(* IEC 61131-3 sources: SmartHomeNew/ (part 14) *)

(* ---- PRG_Output_Freshness_Governor.st ---- *)
PROGRAM PRG_Output_Freshness_Governor
VAR
    L_Now_MS : UDINT;
    L_Delta_MS : UDINT;
    L_Output_Valid : BOOL := TRUE;
    L_Error_Code : UDINT := 0;
    L_Error_Text : STRING(160) := '';
END_VAR

L_Now_MS := GVL_STATUS.G_System_Time_MS;
L_Output_Valid := TRUE;
L_Error_Code := 0;
L_Error_Text := '';

IF NOT GVL_RUNTIME_EPOCH.Runtime_Runtime_Barrier_OK THEN
    L_Output_Valid := FALSE;
    L_Error_Code := 6000;
    L_Error_Text := 'Output runtime authority invalid';
END_IF;

IF L_Output_Valid AND (NOT GVL_RUNTIME_EPOCH.Runtime_IO_Publication_Allowed) THEN
    L_Output_Valid := FALSE;
    L_Error_Code := 6001;
    L_Error_Text := 'Output publication not allowed';
END_IF;

IF L_Output_Valid AND (NOT GVL_RUNTIME_SNAPSHOT.Snapshot_Frozen) THEN
    L_Output_Valid := FALSE;
    L_Error_Code := 6100;
    L_Error_Text := 'Runtime snapshot not frozen';
END_IF;

IF L_Output_Valid AND (NOT GVL_RUNTIME_SNAPSHOT.Snapshot_Publication_Allowed) THEN
    L_Output_Valid := FALSE;
    L_Error_Code := 6101;
    L_Error_Text := 'Snapshot publication blocked';
END_IF;

IF L_Output_Valid AND (NOT GVL_RUNTIME_SNAPSHOT.Snapshot_Copy_Valid) THEN
    L_Output_Valid := FALSE;
    L_Error_Code := 6102;
    L_Error_Text := 'Snapshot copy invalid';
END_IF;

IF L_Output_Valid AND (NOT GVL_RUNTIME_SNAPSHOT.Snapshot_Isolation_Valid) THEN
    L_Output_Valid := FALSE;
    L_Error_Code := 6103;
    L_Error_Text := 'Snapshot isolation invalid';
END_IF;

IF L_Output_Valid AND GVL_RUNTIME_SNAPSHOT.Snapshot_Mutation_Detected THEN
    L_Output_Valid := FALSE;
    L_Error_Code := 6104;
    L_Error_Text := 'Snapshot mutation detected';
END_IF;

IF L_Output_Valid AND GVL_DISTRIBUTED_EPOCH.Distributed_Quarantine_Active THEN
    L_Output_Valid := FALSE;
    L_Error_Code := 6200;
    L_Error_Text := 'Distributed reconciliation quarantine active';
END_IF;

IF L_Output_Valid AND (NOT GVL_DISTRIBUTED_SNAPSHOT.Distributed_Publication_Reconciled) THEN
    L_Output_Valid := FALSE;
    L_Error_Code := 6300;
    L_Error_Text := 'Distributed publication reconciliation invalid';
END_IF;

IF L_Output_Valid AND (NOT GVL_DISTRIBUTED_SNAPSHOT.Distributed_Publication_Freeze_Valid) THEN
    L_Output_Valid := FALSE;
    L_Error_Code := 6301;
    L_Error_Text := 'Distributed publication freeze invalid';
END_IF;

IF L_Output_Valid AND (NOT GVL_DISTRIBUTED_SNAPSHOT.Distributed_Snapshot_Consistent) THEN
    L_Output_Valid := FALSE;
    L_Error_Code := 6302;
    L_Error_Text := 'Distributed immutable snapshot inconsistent';
END_IF;

IF L_Output_Valid AND GVL_DISTRIBUTED_SNAPSHOT.Distributed_Snapshot_Quarantine_Active THEN
    L_Output_Valid := FALSE;
    L_Error_Code := 6306;
    L_Error_Text := 'Distributed immutable snapshot quarantine active';
END_IF;

// Finalized distributed publication continuity.
IF L_Output_Valid AND (NOT GVL_DISTRIBUTED_COMMIT.Distributed_Commit_Valid) THEN
    L_Output_Valid := FALSE;
    L_Error_Code := 6400;
    L_Error_Text := 'Distributed commit invalid';
END_IF;

IF L_Output_Valid AND (NOT GVL_DISTRIBUTED_COMMIT.Publication_Prepare_Valid) THEN
    L_Output_Valid := FALSE;
    L_Error_Code := 6402;
    L_Error_Text := 'Distributed publication prepare invalid';
END_IF;

IF L_Output_Valid AND GVL_DISTRIBUTED_COMMIT.Publication_Commit_Requested
   AND (NOT GVL_DISTRIBUTED_COMMIT.Publication_Commit_Confirmed) THEN
    L_Output_Valid := FALSE;
    L_Error_Code := 6403;
    L_Error_Text := 'Distributed publication commit pending';
END_IF;

IF L_Output_Valid AND GVL_DISTRIBUTED_COMMIT.Peer_Commit_Mismatch THEN
    L_Output_Valid := FALSE;
    L_Error_Code := 6404;
    L_Error_Text := 'Distributed peer commit mismatch';
END_IF;

IF L_Output_Valid AND GVL_DISTRIBUTED_COMMIT.Distributed_Commit_Quarantine_Active THEN
    L_Output_Valid := FALSE;
    L_Error_Code := 6401;
    L_Error_Text := 'Distributed commit quarantine active';
END_IF;

IF L_Output_Valid AND GVL_DISTRIBUTED_COMMIT.Commit_Lease_Expired THEN
    L_Output_Valid := FALSE;
    L_Error_Code := 6405;
    L_Error_Text := 'Distributed commit lease expired';
END_IF;

GVL_OUTPUT_EPOCH.Output_Semantic_Continuity_Warning :=
    (NOT GVL_SEMANTIC_PROGRESS.Semantic_Forward_Progress_Valid)
    OR (NOT GVL_SEMANTIC_PROGRESS.Semantic_Execution_Continuity_OK)
    OR GVL_SEMANTIC_PROGRESS.Semantic_Stagnation_Detected
    OR GVL_SEMANTIC_PROGRESS.Semantic_Replay_Suspected
    OR GVL_SEMANTIC_PROGRESS.Semantic_Livelock_Suspected
    OR GVL_SEMANTIC_PROGRESS.Semantic_Deadlock_Suspected
    OR GVL_SEMANTIC_PROGRESS.Semantic_Progress_Lease_Expired
    OR GVL_SEMANTIC_PROGRESS.Semantic_Progress_Quarantine_Active;

IF L_Output_Valid THEN
    IF GVL_OUTPUT_EPOCH.Output_Runtime_Epoch > GVL_RUNTIME_EPOCH.Runtime_Epoch THEN
        L_Output_Valid := FALSE;
        L_Error_Code := 6002;
        L_Error_Text := 'Output epoch ahead of runtime epoch';
    END_IF;
END_IF;

L_Delta_MS := L_Now_MS - GVL_OUTPUT_EPOCH.Output_Last_Refresh_MS;

IF L_Output_Valid AND GVL_OUTPUT_EPOCH.Output_Lease_Active THEN
    IF L_Delta_MS > GVL_OUTPUT_EPOCH.Output_Lease_Timeout_MS THEN
        L_Output_Valid := FALSE;
        L_Error_Code := 6003;
        L_Error_Text := 'Output lease expired';
    END_IF;
END_IF;

IF L_Output_Valid THEN
    GVL_OUTPUT_EPOCH.Output_Publication_Epoch := GVL_OUTPUT_EPOCH.Output_Publication_Epoch + 1;

    GVL_OUTPUT_EPOCH.Output_Publication_Valid := TRUE;
    GVL_OUTPUT_EPOCH.Output_Lease_Active := TRUE;
    GVL_OUTPUT_EPOCH.Output_Lease_Expired := FALSE;

    GVL_OUTPUT_EPOCH.Output_Runtime_Epoch := GVL_RUNTIME_EPOCH.Runtime_Epoch;
    GVL_OUTPUT_EPOCH.Output_Runtime_Epoch_Valid := TRUE;

    GVL_OUTPUT_EPOCH.Output_Last_Publication_MS := L_Now_MS;
    GVL_OUTPUT_EPOCH.Output_Last_Refresh_MS := L_Now_MS;

    IF GVL_CONVERGENCE.Convergence_Release_Allowed THEN
        GVL_OUTPUT_EPOCH.Output_Stale_Detected := FALSE;
        GVL_OUTPUT_EPOCH.Output_Forced_Safe_Decay := FALSE;
    END_IF;

    GVL_OUTPUT_EPOCH.Output_Last_Error_Code := 0;
    GVL_OUTPUT_EPOCH.Output_Last_Error_Text := '';
ELSE
    GVL_OUTPUT_EPOCH.Output_Publication_Valid := FALSE;
    GVL_OUTPUT_EPOCH.Output_Lease_Expired := TRUE;
    GVL_OUTPUT_EPOCH.Output_Stale_Detected := TRUE;
    GVL_OUTPUT_EPOCH.Output_Forced_Safe_Decay := TRUE;

    GVL_OUTPUT_EPOCH.Output_Last_Invalidation_MS := L_Now_MS;
    GVL_OUTPUT_EPOCH.Output_Last_Error_Code := L_Error_Code;
    GVL_OUTPUT_EPOCH.Output_Last_Error_Text := L_Error_Text;
END_IF;
END_PROGRAM

(* ---- PRG_Peer_Session_Publication.st ---- *)
PROGRAM PRG_Peer_Session_Publication
// ======================================================
// PEER SESSION PUBLICATION
// ======================================================
// Canonical local PLC session export.
//
// Purpose:
// publish normalized runtime/session authority state into
// explicit peer-session transport contract surface.
//
// This layer does NOT:
// - perform network replication
// - perform distributed reconciliation
// - consume remote peer state
//
// Future transport/replication layers may replicate these
// fields to partner PLCs or external HA channels.
// ======================================================

GVL_PEER_SESSION.Remote_Session_Valid :=
    GVL_RUNTIME_EPOCH.Runtime_IO_Publication_Allowed;

GVL_PEER_SESSION.Remote_Last_Refresh_MS :=
    GVL_STATUS.G_System_Time_MS;

GVL_PEER_SESSION.Remote_Runtime_Epoch :=
    GVL_RUNTIME_EPOCH.Runtime_Epoch;

GVL_PEER_SESSION.Remote_Snapshot_Epoch :=
    GVL_RUNTIME_SNAPSHOT.Snapshot_Epoch;

GVL_PEER_SESSION.Remote_Boot_Generation :=
    GVL_TIME_MONOTONIC.Boot_Generation_ID;

GVL_PEER_SESSION.Remote_Fencing_Token :=
    GVL_PLC_FENCING.PLC_Fencing_Token;

GVL_PEER_SESSION.Remote_Publication_Allowed :=
    GVL_OUTPUT_EPOCH.Output_Publication_Allowed;

GVL_PEER_SESSION.Remote_Runtime_Healthy :=
    GVL_RUNTIME_EPOCH.Runtime_Healthy;

// >>> BULK_SYNC_ANCHOR: PRG_Peer_Session_Publication <<<
END_PROGRAM

(* ---- PRG_Physical_Deadlock_Resolution_Governor.st ---- *)
PROGRAM PRG_Physical_Deadlock_Resolution_Governor
IF GVL_ENERGY_RESURRECTION_BOUNDARY_FABRIC.Energy_Resurrection_Boundary_Granted
AND NOT GVL_PHYSICAL_DEADLOCK_RESOLUTION_FABRIC.Physical_CircularWait_Detected
AND NOT GVL_PHYSICAL_DEADLOCK_RESOLUTION_FABRIC.CrossDomain_Progress_Deadlock
AND NOT GVL_PHYSICAL_DEADLOCK_RESOLUTION_FABRIC.Recovery_Livelock_Detected
AND NOT GVL_PHYSICAL_DEADLOCK_RESOLUTION_FABRIC.Physical_Progress_Stall_Detected THEN

    GVL_PHYSICAL_DEADLOCK_RESOLUTION_FABRIC.Physical_Deadlock_Resolution_Valid := TRUE;
    GVL_PHYSICAL_DEADLOCK_RESOLUTION_FABRIC.Physical_Deadlock_Resolution_Granted := TRUE;
    GVL_PHYSICAL_DEADLOCK_RESOLUTION_FABRIC.Deadlock_Resolution_Canonical := TRUE;
    GVL_PHYSICAL_DEADLOCK_RESOLUTION_FABRIC.Physical_Forward_Progress_Valid := TRUE;
    GVL_PHYSICAL_DEADLOCK_RESOLUTION_FABRIC.CrossDomain_Execution_Progress_Stable := TRUE;
END_IF;
END_PROGRAM

(* ---- PRG_Physical_Reality_Validation_Governor.st ---- *)
PROGRAM PRG_Physical_Reality_Validation_Governor
// PASSIVE PHYSICS REALITY VERIFICATION
// NO EXECUTION MUTATION
// NO ACTUATION MUTATION
// NO AUTHORITY MUTATION

GVL_PHYSICAL_REALITY_VERIFICATION_FABRIC.Physical_Runtime_Reality_Valid :=
    GVL_OPERATIONAL_INTELLIGENCE_FABRIC.Runtime_Causal_Projection_Valid;

GVL_PHYSICAL_REALITY_VERIFICATION_FABRIC.Commanded_State_Verified_Physically :=
    GVL_RUNTIME_TRANSITION_SYSTEM.Runtime_Transition_Legal;

GVL_PHYSICAL_REALITY_VERIFICATION_FABRIC.Physical_Response_Coherent :=
    GVL_TEMPORAL_CAUSALITY_CLOSURE_FABRIC.Temporal_Causality_Coherent;

GVL_PHYSICAL_REALITY_VERIFICATION_FABRIC.Sensor_Physics_Coherent := TRUE;

IF GVL_RUNTIME_TRANSITION_SYSTEM.Illegal_Runtime_Transition_Observed THEN
    GVL_PHYSICAL_REALITY_VERIFICATION_FABRIC.Physical_Reality_Divergence_Detected := TRUE;
END_IF;

IF GVL_RUNTIME_TRANSITION_SYSTEM.Unsafe_State_Promotion_Observed THEN
    GVL_PHYSICAL_REALITY_VERIFICATION_FABRIC.Commanded_State_Mismatch_Detected := TRUE;
END_IF;

IF GVL_TEMPORAL_CAUSALITY_CLOSURE_FABRIC.Temporal_Fork_Detected THEN
    GVL_PHYSICAL_REALITY_VERIFICATION_FABRIC.Impossible_Physical_Response_Detected := TRUE;
END_IF;

END_PROGRAM

(* ---- PRG_Physical_SafeState_Lattice_Governor.st ---- *)
PROGRAM PRG_Physical_SafeState_Lattice_Governor
VAR
    L_Now_MS : UDINT;
    L_Valid : BOOL := TRUE;
END_VAR

L_Now_MS := GVL_STATUS.G_System_Time_MS;

GVL_PHYSICAL_SAFESTATE_LATTICE_FABRIC.Physical_SafeState_Lattice_Valid := FALSE;
GVL_PHYSICAL_SAFESTATE_LATTICE_FABRIC.Physical_SafeState_Lattice_Granted := FALSE;
GVL_PHYSICAL_SAFESTATE_LATTICE_FABRIC.Physical_SafeState_Lattice_Quarantine_Active := TRUE;

IF NOT GVL_GOVERNANCE_PUBLICATION_BINDING_FABRIC.Governance_Publication_Binding_Granted THEN
    L_Valid := FALSE;
END_IF;

IF GVL_PHYSICAL_SAFESTATE_LATTICE_FABRIC.SafeState_Ambiguity_Detected
OR GVL_PHYSICAL_SAFESTATE_LATTICE_FABRIC.Partial_SafeState_Asymmetry_Detected
OR GVL_PHYSICAL_SAFESTATE_LATTICE_FABRIC.Physical_SafeState_Deadlock_Detected
OR GVL_PHYSICAL_SAFESTATE_LATTICE_FABRIC.Unsafe_SafeState_Topology_Detected
OR GVL_PHYSICAL_SAFESTATE_LATTICE_FABRIC.Residual_Unsafe_Actuation_Detected
OR GVL_PHYSICAL_SAFESTATE_LATTICE_FABRIC.SafeState_Energy_Leakage_Detected THEN
    L_Valid := FALSE;
END_IF;

IF L_Valid THEN
    GVL_PHYSICAL_SAFESTATE_LATTICE_FABRIC.Physical_SafeState_Lattice_Valid := TRUE;
    GVL_PHYSICAL_SAFESTATE_LATTICE_FABRIC.Physical_SafeState_Lattice_Granted := TRUE;
    GVL_PHYSICAL_SAFESTATE_LATTICE_FABRIC.Physical_SafeState_Lattice_Quarantine_Active := FALSE;

    GVL_PHYSICAL_SAFESTATE_LATTICE_FABRIC.Canonical_SafeState_Topology_Valid := TRUE;
    GVL_PHYSICAL_SAFESTATE_LATTICE_FABRIC.Physical_SafeState_Lattice_Coherent := TRUE;
    GVL_PHYSICAL_SAFESTATE_LATTICE_FABRIC.Deterministic_FailSafe_Convergence_Granted := TRUE;

    GVL_PHYSICAL_SAFESTATE_LATTICE_FABRIC.Physical_SafeState_Lattice_Epoch :=
        GVL_GOVERNANCE_PUBLICATION_BINDING_FABRIC.Governance_Publication_Binding_Epoch;

    GVL_PHYSICAL_SAFESTATE_LATTICE_FABRIC.Physical_SafeState_Lattice_Epoch_Coherent := TRUE;
    GVL_PHYSICAL_SAFESTATE_LATTICE_FABRIC.Physical_SafeState_Lattice_Last_Update_MS := L_Now_MS;
    GVL_PHYSICAL_SAFESTATE_LATTICE_FABRIC.Physical_SafeState_Lattice_Lease_Expired := FALSE;
END_IF;

END_PROGRAM

(* ---- PRG_Physical_Snapshot_Governor.st ---- *)
PROGRAM PRG_Physical_Snapshot_Governor
VAR
    L_Now_MS : UDINT;
    L_Snapshot_Valid : BOOL := TRUE;
    L_Error_Code : UDINT := 0;
    L_Error_Text : STRING(160) := '';
END_VAR

L_Now_MS := GVL_STATUS.G_System_Time_MS;
L_Snapshot_Valid := TRUE;
L_Error_Code := 0;
L_Error_Text := '';

GVL_PHYSICAL_SNAPSHOT.Physical_Snapshot_Valid := FALSE;
GVL_PHYSICAL_SNAPSHOT.Physical_Snapshot_Frozen := FALSE;
GVL_PHYSICAL_SNAPSHOT.Physical_Snapshot_Publication_Allowed := FALSE;
GVL_PHYSICAL_SNAPSHOT.Physical_Snapshot_Isolation_Valid := FALSE;
GVL_PHYSICAL_SNAPSHOT.Physical_Snapshot_Copy_Valid := FALSE;
GVL_PHYSICAL_SNAPSHOT.Physical_Snapshot_Freshness_Valid := FALSE;
GVL_PHYSICAL_SNAPSHOT.Physical_Snapshot_Consensus_Coherent := FALSE;
GVL_PHYSICAL_SNAPSHOT.Physical_Snapshot_Causality_Coherent := FALSE;

GVL_PHYSICAL_SNAPSHOT.Physical_Snapshot_Runtime_Epoch := ULINT_TO_UDINT(GVL_RUNTIME_EPOCH.Runtime_Epoch);
GVL_PHYSICAL_SNAPSHOT.Physical_Snapshot_Output_Epoch := ULINT_TO_UDINT(GVL_OUTPUT_EPOCH.Output_Publication_Epoch);

IF NOT GVL_RUNTIME_EPOCH.Runtime_Runtime_Barrier_OK THEN
    L_Snapshot_Valid := FALSE;
    L_Error_Code := 23000;
    L_Error_Text := 'Physical snapshot runtime barrier invalid';
END_IF;

IF L_Snapshot_Valid AND NOT GVL_OUTPUT_EPOCH.Output_Publication_Valid THEN
    L_Snapshot_Valid := FALSE;
    L_Error_Code := 23001;
    L_Error_Text := 'Physical snapshot output publication invalid';
END_IF;

IF L_Snapshot_Valid AND GVL_PHYSICAL_SNAPSHOT.Physical_Snapshot_Mutation_Detected THEN
    L_Snapshot_Valid := FALSE;
    L_Error_Code := 23002;
    L_Error_Text := 'Physical snapshot mutation detected';
END_IF;

IF L_Snapshot_Valid AND GVL_PHYSICAL_SNAPSHOT.Physical_Snapshot_Replay_Suspected THEN
    L_Snapshot_Valid := FALSE;
    L_Error_Code := 23003;
    L_Error_Text := 'Physical snapshot replay suspected';
END_IF;

IF L_Snapshot_Valid AND GVL_PHYSICAL_SNAPSHOT.Physical_Snapshot_Lease_Expired THEN
    L_Snapshot_Valid := FALSE;
    L_Error_Code := 23004;
    L_Error_Text := 'Physical snapshot lease expired';
END_IF;

IF L_Snapshot_Valid THEN
    GVL_PHYSICAL_SNAPSHOT.Physical_Snapshot_Valid := TRUE;
    GVL_PHYSICAL_SNAPSHOT.Physical_Snapshot_Frozen := TRUE;
    GVL_PHYSICAL_SNAPSHOT.Physical_Snapshot_Publication_Allowed := TRUE;
    GVL_PHYSICAL_SNAPSHOT.Physical_Snapshot_Isolation_Valid := TRUE;
    GVL_PHYSICAL_SNAPSHOT.Physical_Snapshot_Copy_Valid := TRUE;
    GVL_PHYSICAL_SNAPSHOT.Physical_Snapshot_Freshness_Valid := TRUE;
    GVL_PHYSICAL_SNAPSHOT.Physical_Snapshot_Consensus_Coherent := TRUE;
    GVL_PHYSICAL_SNAPSHOT.Physical_Snapshot_Causality_Coherent := TRUE;
    GVL_PHYSICAL_SNAPSHOT.Physical_Snapshot_Epoch := GVL_PHYSICAL_SNAPSHOT.Physical_Snapshot_Epoch + 1;
    GVL_PHYSICAL_SNAPSHOT.Physical_Snapshot_Last_Update_MS := L_Now_MS;
    GVL_PHYSICAL_SNAPSHOT.Physical_Snapshot_Last_Error_Code := 0;
    GVL_PHYSICAL_SNAPSHOT.Physical_Snapshot_Last_Error_Text := '';
ELSE
    GVL_PHYSICAL_SNAPSHOT.Physical_Snapshot_Valid := FALSE;
    GVL_PHYSICAL_SNAPSHOT.Physical_Snapshot_Frozen := FALSE;
    GVL_PHYSICAL_SNAPSHOT.Physical_Snapshot_Publication_Allowed := FALSE;
    GVL_PHYSICAL_SNAPSHOT.Physical_Snapshot_Last_Error_Code := L_Error_Code;
    GVL_PHYSICAL_SNAPSHOT.Physical_Snapshot_Last_Error_Text := L_Error_Text;
    GVL_PHYSICAL_SNAPSHOT.Physical_Snapshot_Invalidation_Count := GVL_PHYSICAL_SNAPSHOT.Physical_Snapshot_Invalidation_Count + 1;
END_IF;

END_PROGRAM

(* ---- PRG_PLC_Arbitration.st ---- *)
PROGRAM PRG_PLC_Arbitration
// Local-only PLC authority for the cold-spare architecture.
//
// Hot A/B failover and lowest-ID arbitration are intentionally disabled.
// The reserve PLC is not expected to be connected to the same physical outputs
// during normal runtime.

GVL_STATUS.G_Is_Active_PLC := TRUE;
GVL_STATUS.G_Other_PLC_Is_Active := FALSE;
GVL_STATUS.G_Remote_PLC_Alive := FALSE;
GVL_STATUS.G_Active_PLC_ID := GVL_STATUS.G_Local_PLC_ID;

// Keep remote visibility fields reset so old partner pulses cannot resurrect a
// standby/active split-brain path.
GVL_STATUS.G_Remote_PLC_Pulse := FALSE;
GVL_STATUS.G_Remote_PLC_Last_Seen_MS := 0;

// >>> BULK_SYNC_ANCHOR: PRG_PLC_Arbitration <<<
END_PROGRAM

(* ---- PRG_PLC_Fencing_Governor.st ---- *)
PROGRAM PRG_PLC_Fencing_Governor
VAR
    L_Now_MS : UDINT;
END_VAR

L_Now_MS := GVL_STATUS.G_System_Time_MS;

// ======================================================
// LOCAL-ONLY PLC FENCING GOVERNOR
// ======================================================
// Cold-spare architecture: there is exactly one runtime owner.
// A reserve PLC is not connected in parallel and is not allowed to arbitrate
// outputs during normal runtime. Therefore split-brain/stale-owner detection is
// held inactive here while still publishing a valid local ownership epoch/token
// for downstream authority checks.
// ======================================================

GVL_PLC_FENCING.PLC_Heartbeat_Only_Mode := FALSE;
GVL_PLC_FENCING.PLC_Split_Brain_Detected := FALSE;
GVL_PLC_FENCING.PLC_Stale_Owner_Detected := FALSE;
GVL_PLC_FENCING.PLC_Asymmetric_Partition_Detected := FALSE;
GVL_PLC_FENCING.PLC_Forced_Safe_Quarantine := FALSE;

GVL_PLC_FENCING.PLC_Ownership_Epoch := GVL_PLC_FENCING.PLC_Ownership_Epoch + 1;
GVL_PLC_FENCING.PLC_Fencing_Token := GVL_PLC_FENCING.PLC_Ownership_Epoch;

GVL_PLC_FENCING.PLC_Ownership_Valid := TRUE;
GVL_PLC_FENCING.PLC_Semantic_Authority_Valid := TRUE;

GVL_PLC_FENCING.PLC_Lease_Active := TRUE;
GVL_PLC_FENCING.PLC_Lease_Expired := FALSE;
GVL_PLC_FENCING.PLC_Last_Lease_Refresh_MS := L_Now_MS;
GVL_PLC_FENCING.PLC_Last_Authority_Validation_MS := L_Now_MS;

GVL_PLC_FENCING.PLC_Last_Error_Code := 0;
GVL_PLC_FENCING.PLC_Last_Error_Text := '';

// >>> BULK_SYNC_ANCHOR: PRG_PLC_Fencing_Governor <<<
END_PROGRAM

(* ---- PRG_Policy.st ---- *)
PROGRAM PRG_Policy
VAR
    L_Away_Elapsed_MS : UDINT;
    L_Restore_Elapsed_MS : UDINT;
    L_Return_Delta_MS : UDINT;
    L_Return_Grace_Elapsed_MS : UDINT;
    L_Away_Return_Window_Reached : BOOL;
    L_Previous_Away_Active : BOOL := FALSE;
    L_Previous_Away_Level : BYTE := 0;
END_VAR

GVL_POLICY.G_Away_Restore_Requested := FALSE;

// ============================================================
// CONFIGURATION SAFETY CLAMP
// ============================================================
// Configuration validation is diagnostic-only here.
// System mode ownership remains in FB_State_Manager via
// FB_System_Health_Orchestrator. Policy must not directly write
// GVL_STATE.G_System_Mode.
IF GVL_CONFIG_VALIDATION.G_Config_Force_Safe_Mode AND
   (NOT GVL_CONFIG_VALIDATION.G_Config_Valid) AND
   (GVL_STATE.G_System_Mode = E_System_Operating_Mode.MODE_NORMAL) THEN
    GVL_STATUS.G_Diagnostics.Subsystem_Degraded := TRUE;
    GVL_STATUS.G_System_Mode_Text := 'CONFIG DEGRADED';
END_IF;

// ============================================================
// SCENARIO POLICY OWNER
// ============================================================

// 1. Base priority resolution
IF GVL_STATE.G_System_Mode = E_System_Operating_Mode.MODE_SAFE_STOP THEN
    GVL_POLICY.G_Scenario_Intent := E_SCENARIO_TYPE.SCENARIO_NONE;
    GVL_POLICY.G_Scenario_Source := SRC_SAFETY;

ELSIF GVL_POLICY.G_Scenario_Request_Operator <> E_SCENARIO_TYPE.SCENARIO_NONE THEN
    GVL_POLICY.G_Scenario_Intent := GVL_POLICY.G_Scenario_Request_Operator;
    GVL_POLICY.G_Scenario_Source := SRC_OPERATOR;

ELSIF GVL_POLICY.G_Scenario_Request_Gateway <> E_SCENARIO_TYPE.SCENARIO_NONE THEN
    GVL_POLICY.G_Scenario_Intent := GVL_POLICY.G_Scenario_Request_Gateway;
    GVL_POLICY.G_Scenario_Source := SRC_GATEWAY;

ELSIF GVL_POLICY.G_Scenario_Request_Rule <> E_SCENARIO_TYPE.SCENARIO_NONE THEN
    GVL_POLICY.G_Scenario_Intent := GVL_POLICY.G_Scenario_Request_Rule;
    GVL_POLICY.G_Scenario_Source := SRC_RULE;

ELSE
    GVL_POLICY.G_Scenario_Intent := GVL_STATUS.G_Current_Scenario;
    GVL_POLICY.G_Scenario_Source := SRC_NONE;
END_IF;

// 2. Fail-safe clamp
CASE GVL_STATE.G_System_Mode OF
    E_System_Operating_Mode.MODE_SAFE_STOP:
        GVL_POLICY.G_Scenario_Intent := E_SCENARIO_TYPE.SCENARIO_NONE;
        GVL_POLICY.G_Scenario_Source := SRC_SAFETY;

    E_System_Operating_Mode.MODE_FREEZE_PROTECTION:
        GVL_POLICY.G_Scenario_Intent := E_SCENARIO_TYPE.SCENARIO_NONE;
        GVL_POLICY.G_Scenario_Source := SRC_POLICY;

    E_System_Operating_Mode.MODE_DEGRADED:
        CASE GVL_POLICY.G_Scenario_Intent OF
            E_SCENARIO_TYPE.SCENARIO_NONE,
            E_SCENARIO_TYPE.SCENARIO_PRESENCE,
            E_SCENARIO_TYPE.SCENARIO_AWAY,
            E_SCENARIO_TYPE.SCENARIO_SLEEP:
                ;
        ELSE
            GVL_POLICY.G_Scenario_Intent := E_SCENARIO_TYPE.SCENARIO_NONE;
            GVL_POLICY.G_Scenario_Source := SRC_POLICY;
        END_CASE;
END_CASE;

// 3. Context automation
IF GVL_STATE.G_System_Mode = E_System_Operating_Mode.MODE_NORMAL THEN
    IF GVL_ALARM.G_Security_Armed AND
       (GVL_POLICY.G_Scenario_Request_Operator = E_SCENARIO_TYPE.SCENARIO_NONE) AND
       (GVL_POLICY.G_Scenario_Request_Gateway = E_SCENARIO_TYPE.SCENARIO_NONE) AND
       (GVL_POLICY.G_Scenario_Request_Rule = E_SCENARIO_TYPE.SCENARIO_NONE) AND
       (GVL_POLICY.G_Scenario_Intent <> E_SCENARIO_TYPE.SCENARIO_AWAY) THEN
        GVL_POLICY.G_Scenario_Intent := E_SCENARIO_TYPE.SCENARIO_AWAY;
        GVL_POLICY.G_Scenario_Source := SRC_POLICY;
    END_IF;
END_IF;

// 4. Degraded adaptation
IF GVL_STATE.G_System_Mode = E_System_Operating_Mode.MODE_DEGRADED THEN
    IF (GVL_POLICY.G_Scenario_Request_Operator = E_SCENARIO_TYPE.SCENARIO_NONE) AND
       (GVL_POLICY.G_Scenario_Request_Gateway = E_SCENARIO_TYPE.SCENARIO_NONE) AND
       (GVL_POLICY.G_Scenario_Request_Rule = E_SCENARIO_TYPE.SCENARIO_NONE) THEN

        IF GVL_ALARM.G_Security_Armed THEN
            GVL_POLICY.G_Scenario_Intent := E_SCENARIO_TYPE.SCENARIO_AWAY;
            GVL_POLICY.G_Scenario_Source := SRC_POLICY;

        ELSIF GVL_POLICY.G_Scenario_Intent = E_SCENARIO_TYPE.SCENARIO_PRESENCE THEN
            GVL_POLICY.G_Scenario_Intent := E_SCENARIO_TYPE.SCENARIO_SLEEP;
            GVL_POLICY.G_Scenario_Source := SRC_POLICY;
        END_IF;
    END_IF;
END_IF;

// ============================================================
// AWAY LEVEL POLICY
// ============================================================
// 0=none, 1=short, 2=medium, 3=long.
// Short: light 100%, heating -1C, simulation off.
// Medium: light/simulation medium, heating -3C, simulation 0.3.
// Long: minimal reasonable heating economy; planned-return preheat may
// temporarily raise selected rooms before the expected arrival.
L_Away_Return_Window_Reached := FALSE;

IF GVL_POLICY.G_Scenario_Intent = E_SCENARIO_TYPE.SCENARIO_AWAY THEN
    IF NOT GVL_POLICY.G_Away_Active THEN
        GVL_POLICY.G_Away_Active := TRUE;
        GVL_POLICY.G_Away_Start_MS := GVL_TIME_SERVICE.G_Now_MS;
        GVL_POLICY.G_Away_Elapsed_MS := 0;
        GVL_POLICY.G_Away_Level := 1;
        GVL_POLICY.G_Away_Return_Preheat_Active := FALSE;
        GVL_POLICY.G_Away_Return_Grace_Active := FALSE;
        GVL_POLICY.G_Away_Return_Expired := FALSE;
    ELSE
        IF GVL_TIME_SERVICE.G_Now_MS >= GVL_POLICY.G_Away_Start_MS THEN
            L_Away_Elapsed_MS := GVL_TIME_SERVICE.G_Now_MS - GVL_POLICY.G_Away_Start_MS;
        ELSE
            L_Away_Elapsed_MS := (4294967295 - GVL_POLICY.G_Away_Start_MS) + GVL_TIME_SERVICE.G_Now_MS + 1;
        END_IF;

        GVL_POLICY.G_Away_Elapsed_MS := L_Away_Elapsed_MS;

        IF L_Away_Elapsed_MS >= GVL_POLICY.G_Away_Medium_To_Long_MS THEN
            GVL_POLICY.G_Away_Level := 3;
        ELSIF L_Away_Elapsed_MS >= GVL_POLICY.G_Away_Short_To_Medium_MS THEN
            GVL_POLICY.G_Away_Level := 2;
        ELSE
            GVL_POLICY.G_Away_Level := 1;
        END_IF;
    END_IF;

    // Planned return preheat window.
    IF GVL_POLICY.G_Away_Planned_Return_Enabled AND NOT GVL_POLICY.G_Away_Return_Expired THEN
        IF GVL_POLICY.G_Away_Planned_Return_MS >= GVL_TIME_SERVICE.G_Now_MS THEN
            L_Return_Delta_MS := GVL_POLICY.G_Away_Planned_Return_MS - GVL_TIME_SERVICE.G_Now_MS;
            L_Away_Return_Window_Reached := (L_Return_Delta_MS <= GVL_POLICY.G_Away_Preheat_Lead_MS);
        ELSE
            L_Away_Return_Window_Reached := TRUE;
        END_IF;

        IF L_Away_Return_Window_Reached THEN
            GVL_POLICY.G_Away_Return_Preheat_Active := TRUE;

            IF NOT GVL_POLICY.G_Away_Return_Grace_Active THEN
                GVL_POLICY.G_Away_Return_Grace_Active := TRUE;
                GVL_POLICY.G_Away_Return_Grace_Start_MS := GVL_TIME_SERVICE.G_Now_MS;
            END_IF;
        END_IF;

        IF GVL_POLICY.G_Away_Return_Grace_Active THEN
            IF GVL_TIME_SERVICE.G_Now_MS >= GVL_POLICY.G_Away_Return_Grace_Start_MS THEN
                L_Return_Grace_Elapsed_MS := GVL_TIME_SERVICE.G_Now_MS - GVL_POLICY.G_Away_Return_Grace_Start_MS;
            ELSE
                L_Return_Grace_Elapsed_MS := (4294967295 - GVL_POLICY.G_Away_Return_Grace_Start_MS) + GVL_TIME_SERVICE.G_Now_MS + 1;
            END_IF;

            IF L_Return_Grace_Elapsed_MS >= GVL_POLICY.G_Away_Return_Grace_MS THEN
                GVL_POLICY.G_Away_Return_Expired := TRUE;
                GVL_POLICY.G_Away_Return_Preheat_Active := FALSE;
                GVL_POLICY.G_Away_Return_Grace_Active := FALSE;
            END_IF;
        END_IF;
    ELSE
        GVL_POLICY.G_Away_Return_Preheat_Active := FALSE;
        GVL_POLICY.G_Away_Return_Grace_Active := FALSE;
    END_IF;

    CASE GVL_POLICY.G_Away_Level OF
        1:
            GVL_POLICY.G_Away_Simulation_Active := FALSE;
            GVL_POLICY.G_Away_Simulation_Intensity := 0.0;
            GVL_POLICY.G_Away_Heating_Offset_C := -1.0;
        2:
            GVL_POLICY.G_Away_Simulation_Active := TRUE;
            GVL_POLICY.G_Away_Simulation_Intensity := 0.3;
            GVL_POLICY.G_Away_Heating_Offset_C := -3.0;
        3:
            GVL_POLICY.G_Away_Simulation_Active := TRUE;
            GVL_POLICY.G_Away_Simulation_Intensity := 0.2;

            IF GVL_POLICY.G_Away_Return_Preheat_Active THEN
                GVL_POLICY.G_Away_Heating_Offset_C := 0.0;
            ELSE
                GVL_POLICY.G_Away_Heating_Offset_C := GVL_POLICY.G_Away_Long_Economy_Setpoint_C - 22.0;
            END_IF;
    ELSE
            GVL_POLICY.G_Away_Simulation_Active := FALSE;
            GVL_POLICY.G_Away_Simulation_Intensity := 0.0;
            GVL_POLICY.G_Away_Heating_Offset_C := 0.0;
    END_CASE;

ELSE
    IF GVL_POLICY.G_Away_Active AND (GVL_POLICY.G_Away_Level = 1) THEN
        GVL_POLICY.G_Away_Restore_Requested := TRUE;
        GVL_POLICY.G_Away_Restore_Active := TRUE;
        GVL_POLICY.G_Away_Restore_Start_MS := GVL_TIME_SERVICE.G_Now_MS;
    END_IF;

    GVL_POLICY.G_Away_Active := FALSE;
    GVL_POLICY.G_Away_Level := 0;
    GVL_POLICY.G_Away_Elapsed_MS := 0;
    GVL_POLICY.G_Away_Simulation_Active := FALSE;
    GVL_POLICY.G_Away_Simulation_Intensity := 0.0;
    GVL_POLICY.G_Away_Heating_Offset_C := 0.0;
    GVL_POLICY.G_Away_Return_Preheat_Active := FALSE;
    GVL_POLICY.G_Away_Return_Grace_Active := FALSE;
    GVL_POLICY.G_Away_Return_Expired := FALSE;
END_IF;

IF GVL_POLICY.G_Away_Restore_Active THEN
    IF GVL_TIME_SERVICE.G_Now_MS >= GVL_POLICY.G_Away_Restore_Start_MS THEN
        L_Restore_Elapsed_MS := GVL_TIME_SERVICE.G_Now_MS - GVL_POLICY.G_Away_Restore_Start_MS;
    ELSE
        L_Restore_Elapsed_MS := (4294967295 - GVL_POLICY.G_Away_Restore_Start_MS) + GVL_TIME_SERVICE.G_Now_MS + 1;
    END_IF;

    IF L_Restore_Elapsed_MS >= GVL_POLICY.G_Away_Restore_Duration_MS THEN
        GVL_POLICY.G_Away_Restore_Progress := 1.0;
        GVL_POLICY.G_Away_Restore_Active := FALSE;
    ELSE
        GVL_POLICY.G_Away_Restore_Progress := TO_REAL(L_Restore_Elapsed_MS) / TO_REAL(GVL_POLICY.G_Away_Restore_Duration_MS);
    END_IF;
ELSE
    GVL_POLICY.G_Away_Restore_Progress := 0.0;
END_IF;

L_Previous_Away_Active := GVL_POLICY.G_Away_Active;
L_Previous_Away_Level := GVL_POLICY.G_Away_Level;

// 5. Heating bridge
// Policy publishes preheat intent only. Actual per-circuit comfort/economy
// target selection is owned by FB_Heating_Circuit_Control through
// ST_FloorHeating_Circuit_Config.
GVL_STATE.G_Preheat_Request :=
    GVL_POLICY.G_Rule_Preheat_Request OR GVL_POLICY.G_Away_Return_Preheat_Active;
GVL_HEATING_REQUEST.G_Preheat_Request := GVL_STATE.G_Preheat_Request;
GVL_HEATING_REQUEST.G_Target_Temperature := GVL_STATE.G_Target_Temperature;

GVL_STATE.G_Freeze_Request :=
    (GVL_STATE.G_System_Mode = E_System_Operating_Mode.MODE_FREEZE_PROTECTION);
GVL_HEATING_REQUEST.G_Freeze_Request := GVL_STATE.G_Freeze_Request;

PRG_Away_Restore_Manager();
END_PROGRAM

(* ---- PRG_Power_Domain_Segmentation_Governor.st ---- *)
PROGRAM PRG_Power_Domain_Segmentation_Governor
IF GVL_RESIDUAL_ENERGY_STATE_FABRIC.Residual_Energy_State_Valid
AND NOT GVL_POWER_DOMAIN_SEGMENTATION_FABRIC.Unsafe_Power_Resurrection_Detected
AND NOT GVL_POWER_DOMAIN_SEGMENTATION_FABRIC.Partial_Power_Isolation_Asymmetry
AND NOT GVL_POWER_DOMAIN_SEGMENTATION_FABRIC.Distributed_Power_Segmentation_Fork THEN

    GVL_POWER_DOMAIN_SEGMENTATION_FABRIC.Power_Domain_Segmentation_Valid := TRUE;
    GVL_POWER_DOMAIN_SEGMENTATION_FABRIC.Power_Domain_Segmentation_Granted := TRUE;
    GVL_POWER_DOMAIN_SEGMENTATION_FABRIC.Power_Domain_Boundaries_Canonical := TRUE;
    GVL_POWER_DOMAIN_SEGMENTATION_FABRIC.Distributed_Power_Segmentation_Stable := TRUE;
    GVL_POWER_DOMAIN_SEGMENTATION_FABRIC.Power_Reactivation_Isolation_Valid := TRUE;
END_IF;
END_PROGRAM

(* ---- PRG_PreOutput_Safety_Barrier.st ---- *)
PROGRAM PRG_PreOutput_Safety_Barrier
VAR
    L_i : INT;
    L_Now_MS : UDINT;
    L_Block_IO : BOOL := FALSE;
    L_Error_Code : UDINT := 0;
    L_Error_Text : STRING(160) := '';
    L_Any_Manifold_Pump_On : BOOL := FALSE;
    L_Prev_Block_IO : BOOL;

    L_Selective_Projection_Active : BOOL;
    L_Global_Fallback_Active : BOOL;
    L_Runtime_Projection_Healthy : BOOL;

    L_Finalized_Publication_Continuity : BOOL;
    L_Physical_Causality_Healthy : BOOL;
    L_Command_Telemetry_Epoch_Aligned : BOOL;
    L_Physical_Ack_Fresh : BOOL;

    fbLog : FB_LogEvent;
END_VAR

L_Now_MS := GVL_STATUS.G_System_Time_MS;
L_Block_IO := FALSE;
L_Error_Code := 0;
L_Error_Text := '';
L_Any_Manifold_Pump_On := FALSE;
L_Prev_Block_IO := GVL_COMMAND_VERIFY.PreOutput_Block_IO;

L_Selective_Projection_Active :=
    GVL_Water_Isolation_Authority.G_Any_Selective_Authority_Allowed;

L_Global_Fallback_Active :=
    GVL_Water_Isolation_Authority.G_Any_Global_Fallback_Required;

L_Runtime_Projection_Healthy :=
    GVL_Water_Output_Reconciliation.G_Runtime_Valid
    AND NOT GVL_Water_Output_Reconciliation.G_Any_Conflict_Detected;

// Command ↔ telemetry epoch binding.
L_Command_Telemetry_Epoch_Aligned :=
    GVL_TELEMETRY.Command_Epoch = GVL_OUTPUT_EPOCH.Output_Publication_Epoch
    AND GVL_TELEMETRY.Telemetry_Epoch = GVL_OUTPUT_EPOCH.Output_Publication_Epoch
    AND GVL_TELEMETRY.Telemetry_Epoch >=
        GVL_TELEMETRY.Last_Acknowledged_Command_Epoch;

// Physical acknowledgment freshness.
L_Physical_Ack_Fresh :=
    (L_Now_MS - GVL_TELEMETRY.Last_Physical_Ack_Time_MS) <= 5000;

// Physical causality evidence.
L_Physical_Causality_Healthy :=
    GVL_TELEMETRY.Telemetry_Runtime_Valid
    AND GVL_TELEMETRY.Telemetry_Freshness_Valid
    AND NOT GVL_TELEMETRY.Telemetry_Lease_Expired
    AND NOT GVL_TELEMETRY.Telemetry_Quarantine_Active
    AND GVL_TELEMETRY.Command_Telemetry_Causality_Valid
    AND NOT GVL_TELEMETRY.Command_Telemetry_Divergence_Detected
    AND GVL_TELEMETRY.Actuator_Feedback_Valid
    AND GVL_TELEMETRY.Actuator_Feedback_Fresh
    AND GVL_TELEMETRY.Physical_Effect_Confirmed
    AND L_Command_Telemetry_Epoch_Aligned
    AND L_Physical_Ack_Fresh
    AND NOT GVL_TELEMETRY.Telemetry_Replay_Suspected;

// Finalized publication continuity proof chain.
L_Finalized_Publication_Continuity :=
    GVL_SEMANTIC_PROGRESS.Semantic_Forward_Progress_Valid
    AND GVL_SEMANTIC_PROGRESS.Semantic_Execution_Continuity_OK
    AND NOT GVL_SEMANTIC_PROGRESS.Semantic_Stagnation_Detected
    AND NOT GVL_SEMANTIC_PROGRESS.Semantic_Replay_Suspected
    AND NOT GVL_SEMANTIC_PROGRESS.Semantic_Livelock_Suspected
    AND NOT GVL_SEMANTIC_PROGRESS.Semantic_Deadlock_Suspected
    AND NOT GVL_SEMANTIC_PROGRESS.Semantic_Progress_Lease_Expired
    AND NOT GVL_SEMANTIC_PROGRESS.Semantic_Progress_Quarantine_Active
    AND GVL_RUNTIME_SNAPSHOT.Snapshot_Frozen
    AND GVL_RUNTIME_SNAPSHOT.Snapshot_Publication_Allowed
    AND GVL_RUNTIME_SNAPSHOT.Snapshot_Copy_Valid
    AND GVL_RUNTIME_SNAPSHOT.Snapshot_Isolation_Valid
    AND NOT GVL_RUNTIME_SNAPSHOT.Snapshot_Mutation_Detected
    AND GVL_DISTRIBUTED_SNAPSHOT.Distributed_Publication_Reconciled
    AND GVL_DISTRIBUTED_SNAPSHOT.Distributed_Publication_Freeze_Valid
    AND GVL_DISTRIBUTED_SNAPSHOT.Distributed_Snapshot_Consistent
    AND GVL_DISTRIBUTED_COMMIT.Distributed_Commit_Valid
    AND GVL_DISTRIBUTED_COMMIT.Publication_Prepare_Valid
    AND GVL_DISTRIBUTED_COMMIT.Publication_Commit_Confirmed
    AND NOT GVL_DISTRIBUTED_COMMIT.Peer_Commit_Mismatch
    AND NOT GVL_DISTRIBUTED_COMMIT.Distributed_Commit_Quarantine_Active
    AND NOT GVL_DISTRIBUTED_COMMIT.Commit_Lease_Expired
    AND GVL_OUTPUT_EPOCH.Output_Publication_Valid
    AND GVL_OUTPUT_EPOCH.Output_Runtime_Epoch_Valid
    AND NOT GVL_OUTPUT_EPOCH.Output_Lease_Expired
    AND NOT GVL_OUTPUT_EPOCH.Output_Forced_Safe_Decay;

IF (NOT L_Block_IO)
   AND (NOT L_Finalized_Publication_Continuity) THEN
    L_Block_IO := TRUE;
    L_Error_Code := 3999;
    L_Error_Text := 'PreOutput finalized publication continuity invalid';
END_IF;

IF (NOT L_Block_IO)
   AND (NOT L_Physical_Causality_Healthy) THEN
    L_Block_IO := TRUE;
    L_Error_Code := 3998;
    L_Error_Text := 'Physical causality evidence invalid';
END_IF;

IF (NOT L_Block_IO) AND (NOT GVL_STATUS.G_Is_Active_PLC) THEN
    L_Block_IO := TRUE;
    L_Error_Code := 4000;
    L_Error_Text := 'PreOutput inactive PLC';
END_IF;

IF (NOT L_Block_IO)
   AND (GVL_COMMAND.G_Gas_Valve_Close <> GVL_COMMAND_SHADOW.G_Gas_Valve_Close) THEN
    L_Block_IO := TRUE;
    L_Error_Code := 4001;
    L_Error_Text := 'PreOutput gas command mismatch';
END_IF;

IF (NOT L_Block_IO)
   AND (GVL_COMMAND.G_Boiler_Stop <> GVL_COMMAND_SHADOW.G_Boiler_Stop) THEN
    L_Block_IO := TRUE;
    L_Error_Code := 4002;
    L_Error_Text := 'PreOutput boiler command mismatch';
END_IF;

IF (NOT L_Block_IO)
   AND (GVL_COMMAND.G_Vent_Stop <> GVL_COMMAND_SHADOW.G_Vent_Stop) THEN
    L_Block_IO := TRUE;
    L_Error_Code := 4003;
    L_Error_Text := 'PreOutput vent command mismatch';
END_IF;

IF (NOT L_Block_IO)
   AND (GVL_COMMAND.G_Close_Valve_35 <> GVL_COMMAND_SHADOW.G_Close_Valve_35) THEN
    L_Block_IO := TRUE;
    L_Error_Code := 4004;
    L_Error_Text := 'PreOutput valve 35 command mismatch';
END_IF;

IF (NOT L_Block_IO)
   AND (GVL_COMMAND.G_Close_Valve_36 <> GVL_COMMAND_SHADOW.G_Close_Valve_36) THEN
    L_Block_IO := TRUE;
    L_Error_Code := 4005;
    L_Error_Text := 'PreOutput valve 36 command mismatch';
END_IF;

GVL_COMMAND_VERIFY.PreOutput_Physical_Causality_Valid :=
    L_Physical_Causality_Healthy;

GVL_COMMAND_VERIFY.PreOutput_Barrier_OK := NOT L_Block_IO;
GVL_COMMAND_VERIFY.PreOutput_Block_IO := L_Block_IO;
GVL_COMMAND_VERIFY.PreOutput_Last_Error_Code := L_Error_Code;
GVL_COMMAND_VERIFY.PreOutput_Last_Error_Text := L_Error_Text;

IF L_Block_IO THEN
    GVL_COMMAND_VERIFY.PreOutput_Last_Error_Time_MS := L_Now_MS;
    IF NOT L_Prev_Block_IO THEN
        GVL_COMMAND_VERIFY.PreOutput_Block_Count :=
            GVL_COMMAND_VERIFY.PreOutput_Block_Count + 1;
        fbLog(
            VI_Event_Type := 1002,
            VI_Timestamp := L_Now_MS,
            VI_Param1 := L_Error_Code,
            VI_Param2 := GVL_COMMAND_VERIFY.PreOutput_Block_Count
        );
    END_IF;
END_IF;

END_PROGRAM

(* ---- PRG_Presence_Manager.st ---- *)
PROGRAM PRG_Presence_Manager
VAR
    fbPresence : FB_Presence_Manager;
END_VAR

fbPresence(
    VI_Motion_Sensors := GVL_STATE.G_Motion_Sensors,
    VI_System_Time_MS := GVL_STATUS.G_System_Time_MS
);

GVL_PRESENCE.G_Any_Motion := fbPresence.VO_Any_Motion;
GVL_PRESENCE.G_Occupied := fbPresence.VO_Occupied;
GVL_PRESENCE.G_Auto_Away_Request := fbPresence.VO_Auto_Away;
GVL_PRESENCE.G_Last_Motion_TS := fbPresence.VO_Last_Motion_TS;

(* ---- PRG_Provenance_Continuity_Governor.st ---- *)
PROGRAM PRG_Provenance_Continuity_Governor
VAR
    L_Now_MS : UDINT;
    L_Continuity_Valid : BOOL := TRUE;
    L_Error_Code : UDINT := 0;
    L_Error_Text : STRING(160) := '';
END_VAR

L_Now_MS := GVL_STATUS.G_System_Time_MS;
L_Continuity_Valid := TRUE;
L_Error_Code := 0;
L_Error_Text := '';

// Fail-safe defaults.
GVL_PROVENANCE_CONTINUITY_FABRIC.Provenance_Continuity_Valid := FALSE;
GVL_PROVENANCE_CONTINUITY_FABRIC.Provenance_Continuity_Granted := FALSE;
GVL_PROVENANCE_CONTINUITY_FABRIC.Provenance_Continuity_Quarantine_Active := TRUE;

GVL_PROVENANCE_CONTINUITY_FABRIC.Recovery_Provenance_Reattested := FALSE;
GVL_PROVENANCE_CONTINUITY_FABRIC.Authority_Resurrection_Authentic := FALSE;
GVL_PROVENANCE_CONTINUITY_FABRIC.Federation_Rejoin_Provenance_Valid := FALSE;
GVL_PROVENANCE_CONTINUITY_FABRIC.PostRecovery_TrustSeed_Coherent := FALSE;
GVL_PROVENANCE_CONTINUITY_FABRIC.CrossEpoch_Provenance_Continuity_Stable := FALSE;

// Authority provenance required.
IF NOT GVL_AUTHORITY_PROVENANCE_FABRIC.Authority_Provenance_Granted THEN
    L_Continuity_Valid := FALSE;
    L_Error_Code := 47000;
    L_Error_Text := 'Authority provenance not granted';
END_IF;

// Post-recovery provenance bypass detectors.
IF GVL_PROVENANCE_CONTINUITY_FABRIC.Stale_Provenance_Resurrection_Detected THEN
    L_Continuity_Valid := FALSE;
    L_Error_Code := 47001;
    L_Error_Text := 'Stale provenance resurrection detected';
END_IF;

IF GVL_PROVENANCE_CONTINUITY_FABRIC.Recovered_Authority_Without_Reattestation_Detected THEN
    L_Continuity_Valid := FALSE;
    L_Error_Code := 47002;
    L_Error_Text := 'Recovered authority without re-attestation detected';
END_IF;

IF GVL_PROVENANCE_CONTINUITY_FABRIC.Federation_Rejoin_Without_Provenance_Detected THEN
    L_Continuity_Valid := FALSE;
    L_Error_Code := 47003;
    L_Error_Text := 'Federation rejoin without provenance detected';
END_IF;

IF GVL_PROVENANCE_CONTINUITY_FABRIC.CrossEpoch_Trust_Continuity_Broken THEN
    L_Continuity_Valid := FALSE;
    L_Error_Code := 47004;
    L_Error_Text := 'Cross-epoch trust continuity broken';
END_IF;

IF GVL_PROVENANCE_CONTINUITY_FABRIC.Recovery_Trust_Seed_Drift_Detected THEN
    L_Continuity_Valid := FALSE;
    L_Error_Code := 47005;
    L_Error_Text := 'Recovery trust-seed drift detected';
END_IF;

IF GVL_PROVENANCE_CONTINUITY_FABRIC.Provenance_Resurrection_Bypass_Detected THEN
    L_Continuity_Valid := FALSE;
    L_Error_Code := 47006;
    L_Error_Text := 'Provenance resurrection bypass detected';
END_IF;

// Provenance continuity validation.
IF L_Continuity_Valid
AND NOT GVL_PROVENANCE_CONTINUITY_FABRIC.Recovery_Epoch_Authenticity_Valid THEN
    L_Continuity_Valid := FALSE;
    L_Error_Code := 47010;
    L_Error_Text := 'Recovery epoch authenticity invalid';
END_IF;

IF L_Continuity_Valid
AND NOT GVL_PROVENANCE_CONTINUITY_FABRIC.Distributed_Rejoin_Attestation_Coherent THEN
    L_Continuity_Valid := FALSE;
    L_Error_Code := 47011;
    L_Error_Text := 'Distributed rejoin attestation invalid';
END_IF;

IF L_Continuity_Valid
AND NOT GVL_PROVENANCE_CONTINUITY_FABRIC.Authority_Restoration_Provenance_Grounded THEN
    L_Continuity_Valid := FALSE;
    L_Error_Code := 47012;
    L_Error_Text := 'Authority restoration provenance invalid';
END_IF;

IF L_Continuity_Valid
AND NOT GVL_PROVENANCE_CONTINUITY_FABRIC.Provenance_Lease_Continuity_Valid THEN
    L_Continuity_Valid := FALSE;
    L_Error_Code := 47013;
    L_Error_Text := 'Provenance lease continuity invalid';
END_IF;

IF L_Continuity_Valid THEN
    GVL_PROVENANCE_CONTINUITY_FABRIC.Provenance_Continuity_Valid := TRUE;
    GVL_PROVENANCE_CONTINUITY_FABRIC.Provenance_Continuity_Granted := TRUE;
    GVL_PROVENANCE_CONTINUITY_FABRIC.Provenance_Continuity_Quarantine_Active := FALSE;

    GVL_PROVENANCE_CONTINUITY_FABRIC.Recovery_Provenance_Reattested := TRUE;
    GVL_PROVENANCE_CONTINUITY_FABRIC.Authority_Resurrection_Authentic := TRUE;
    GVL_PROVENANCE_CONTINUITY_FABRIC.Federation_Rejoin_Provenance_Valid := TRUE;
    GVL_PROVENANCE_CONTINUITY_FABRIC.PostRecovery_TrustSeed_Coherent := TRUE;
    GVL_PROVENANCE_CONTINUITY_FABRIC.CrossEpoch_Provenance_Continuity_Stable := TRUE;

    GVL_PROVENANCE_CONTINUITY_FABRIC.Provenance_Continuity_Epoch :=
        GVL_AUTHORITY_PROVENANCE_FABRIC.Authority_Provenance_Epoch;

    GVL_PROVENANCE_CONTINUITY_FABRIC.Provenance_Continuity_Epoch_Coherent := TRUE;

    GVL_PROVENANCE_CONTINUITY_FABRIC.Provenance_Continuity_Last_Update_MS :=
        L_Now_MS;

    GVL_PROVENANCE_CONTINUITY_FABRIC.Provenance_Continuity_Lease_Expired := FALSE;

    GVL_PROVENANCE_CONTINUITY_FABRIC.Provenance_Continuity_Last_Error_Code := 0;
    GVL_PROVENANCE_CONTINUITY_FABRIC.Provenance_Continuity_Last_Error_Text := '';
ELSE
    GVL_PROVENANCE_CONTINUITY_FABRIC.Provenance_Continuity_Valid := FALSE;
    GVL_PROVENANCE_CONTINUITY_FABRIC.Provenance_Continuity_Granted := FALSE;
    GVL_PROVENANCE_CONTINUITY_FABRIC.Provenance_Continuity_Quarantine_Active := TRUE;

    GVL_PROVENANCE_CONTINUITY_FABRIC.Provenance_Continuity_Lease_Expired := TRUE;

    GVL_PROVENANCE_CONTINUITY_FABRIC.Provenance_Continuity_Last_Error_Code :=
        L_Error_Code;

    GVL_PROVENANCE_CONTINUITY_FABRIC.Provenance_Continuity_Last_Error_Text :=
        L_Error_Text;

    GVL_PROVENANCE_CONTINUITY_FABRIC.Provenance_Continuity_Invalidation_Count :=
        GVL_PROVENANCE_CONTINUITY_FABRIC.Provenance_Continuity_Invalidation_Count + 1;
END_IF;

END_PROGRAM

(* ---- PRG_Recovery_Cleanup_Governor.st ---- *)
PROGRAM PRG_Recovery_Cleanup_Governor
VAR
    L_Now_MS : UDINT;
    L_Recovery_Valid : BOOL := TRUE;
    L_Error_Code : UDINT := 0;
    L_Error_Text : STRING(160) := '';

    L_Distributed_Recovery_Allowed : BOOL;
    L_Cluster_Recovery_Lock : BOOL;
    L_Cluster_Quarantine : BOOL;
END_VAR

L_Now_MS := GVL_STATUS.G_System_Time_MS;
L_Recovery_Valid := TRUE;
L_Error_Code := 0;
L_Error_Text := '';

// ======================================================
// RECOVERY CLEANUP GOVERNOR
// ======================================================
// Governs cleanup and residue validation after recovery.
//
// Recovery governance is downstream cleanup-oriented.
// It must not feed back into runtime barrier authority.
// Runtime publication authority remains upstream and
// recovery cleanup remains a post-publication residue layer.
//
// Cleanup completion/release is convergence-lease based:
// recovery cleanup is not marked completed/verified on a
// single valid scan.
//
// Distributed recovery governance is authoritative.
// Cleanup/reopen must never bypass:
//   - recovery lock runtime;
//   - cluster quarantine;
//   - centralized recovery execution gates.
// ======================================================

GVL_RECOVERY_GOVERNANCE.Recovery_Semantic_Residue_Detected := FALSE;
GVL_RECOVERY_GOVERNANCE.Recovery_Degraded_State_Residual := FALSE;
GVL_RECOVERY_GOVERNANCE.Recovery_Retained_State_Residual := FALSE;

L_Distributed_Recovery_Allowed :=
    GVL_Distributed_Execution_Gates.G_Can_Recover;

L_Cluster_Recovery_Lock :=
    GVL_Cluster_Runtime_FSM.G_State_Recovery_Lock;

L_Cluster_Quarantine :=
    GVL_Cluster_Runtime_FSM.G_State_Quarantine;

// ------------------------------------------------------
// Monotonic authority linkage.
// ------------------------------------------------------

IF NOT GVL_TIME_MONOTONIC.Monotonic_Time_Valid THEN
    L_Recovery_Valid := FALSE;
    L_Error_Code := 9001;
    L_Error_Text := 'Recovery monotonic authority invalid';
END_IF;

// ------------------------------------------------------
// Distributed recovery governance.
// ------------------------------------------------------

IF L_Recovery_Valid
   AND NOT L_Distributed_Recovery_Allowed THEN

    L_Recovery_Valid := FALSE;

    L_Error_Code := 9010;
    L_Error_Text :=
        'Distributed recovery governance restricted';

END_IF;

// ------------------------------------------------------
// Cluster recovery-lock state.
// ------------------------------------------------------

IF L_Recovery_Valid
   AND L_Cluster_Recovery_Lock THEN

    L_Recovery_Valid := FALSE;

    L_Error_Code := 9011;
    L_Error_Text :=
        'Cluster recovery-lock active';

END_IF;

// ------------------------------------------------------
// Cluster quarantine state.
// ------------------------------------------------------

IF L_Recovery_Valid
   AND L_Cluster_Quarantine THEN

    L_Recovery_Valid := FALSE;

    L_Error_Code := 9012;
    L_Error_Text :=
        'Cluster quarantine active';

END_IF;

// ------------------------------------------------------
// Recovery-active quarantine.
// ------------------------------------------------------

IF GVL_SAFETY_RECOVERY.G_Recovery_Active THEN
    GVL_RECOVERY_GOVERNANCE.Recovery_Quarantine_Active := TRUE;
    GVL_RECOVERY_GOVERNANCE.Recovery_Last_Cleanup_Start_MS := L_Now_MS;

    L_Recovery_Valid := FALSE;

    IF L_Error_Code = 0 THEN
        L_Error_Code := 9002;
        L_Error_Text := 'Recovery quarantine active';
    END_IF;
END_IF;

// ------------------------------------------------------
// Residual degraded-state detection.
// ------------------------------------------------------

IF L_Recovery_Valid AND GVL_DEGRADED.G_System_Degraded THEN
    L_Recovery_Valid := FALSE;
    L_Error_Code := 9003;
    L_Error_Text := 'Residual degraded state detected';

    GVL_RECOVERY_GOVERNANCE.Recovery_Degraded_State_Residual := TRUE;
END_IF;

// ------------------------------------------------------
// Retained-state residue detection.
// ------------------------------------------------------

IF L_Recovery_Valid AND GVL_TIME_MONOTONIC.Retained_Time_Invalid THEN
    L_Recovery_Valid := FALSE;
    L_Error_Code := 9004;
    L_Error_Text := 'Retained state residue detected';

    GVL_RECOVERY_GOVERNANCE.Recovery_Retained_State_Residual := TRUE;
END_IF;

// ------------------------------------------------------
// Publish authoritative recovery governance state.
// ------------------------------------------------------

IF L_Recovery_Valid THEN
    GVL_RECOVERY_GOVERNANCE.Recovery_Epoch := GVL_RECOVERY_GOVERNANCE.Recovery_Epoch + 1;
    GVL_RECOVERY_GOVERNANCE.Recovery_Cleanup_Epoch := GVL_RECOVERY_GOVERNANCE.Recovery_Cleanup_Epoch + 1;

    GVL_RECOVERY_GOVERNANCE.Recovery_Governance_Valid := TRUE;

    // Lease-based cleanup release.
    IF GVL_CONVERGENCE.Convergence_Release_Allowed THEN
        GVL_RECOVERY_GOVERNANCE.Recovery_Cleanup_Completed := TRUE;
        GVL_RECOVERY_GOVERNANCE.Recovery_Cleanup_Verified := TRUE;
        GVL_RECOVERY_GOVERNANCE.Recovery_Quarantine_Active := FALSE;
        GVL_RECOVERY_GOVERNANCE.Recovery_Forced_Safe_Mode := FALSE;
        GVL_RECOVERY_GOVERNANCE.Recovery_Last_Cleanup_End_MS := L_Now_MS;

        GVL_RECOVERY_GOVERNANCE.Recovery_Last_Error_Code := 0;
        GVL_RECOVERY_GOVERNANCE.Recovery_Last_Error_Text := '';
    ELSE
        GVL_RECOVERY_GOVERNANCE.Recovery_Cleanup_Completed := FALSE;
        GVL_RECOVERY_GOVERNANCE.Recovery_Cleanup_Verified := FALSE;
        GVL_RECOVERY_GOVERNANCE.Recovery_Quarantine_Active := TRUE;
        GVL_RECOVERY_GOVERNANCE.Recovery_Forced_Safe_Mode := TRUE;

        GVL_RECOVERY_GOVERNANCE.Recovery_Last_Error_Code := 9005;
        GVL_RECOVERY_GOVERNANCE.Recovery_Last_Error_Text := 'Recovery cleanup waiting for convergence lease';
    END_IF;
ELSE
    // Invalid recovery cleanup state escalates immediately.
    GVL_RECOVERY_GOVERNANCE.Recovery_Governance_Valid := FALSE;
    GVL_RECOVERY_GOVERNANCE.Recovery_Cleanup_Completed := FALSE;
    GVL_RECOVERY_GOVERNANCE.Recovery_Cleanup_Verified := FALSE;

    GVL_RECOVERY_GOVERNANCE.Recovery_Semantic_Residue_Detected := TRUE;
    GVL_RECOVERY_GOVERNANCE.Recovery_Forced_Safe_Mode := TRUE;

    GVL_RECOVERY_GOVERNANCE.Recovery_Last_Error_Code := L_Error_Code;
    GVL_RECOVERY_GOVERNANCE.Recovery_Last_Error_Text := L_Error_Text;

    GVL_RECOVERY_GOVERNANCE.Recovery_Invalidation_Count := GVL_RECOVERY_GOVERNANCE.Recovery_Invalidation_Count + 1;
END_IF;
END_PROGRAM

(* ---- PRG_Recovery_Reactivation_Control_Governor.st ---- *)
PROGRAM PRG_Recovery_Reactivation_Control_Governor
IF GVL_RECOVERY_ORDERING_INTEGRITY_FABRIC.Recovery_Ordering_Integrity_Valid
AND NOT GVL_RECOVERY_REACTIVATION_CONTROL_FABRIC.Unsafe_Reactivation_Ordering_Detected
AND NOT GVL_RECOVERY_REACTIVATION_CONTROL_FABRIC.Partial_Reactivation_Leak_Detected
AND NOT GVL_RECOVERY_REACTIVATION_CONTROL_FABRIC.CrossSubsystem_Reactivation_Fork THEN

    GVL_RECOVERY_REACTIVATION_CONTROL_FABRIC.Recovery_Reactivation_Control_Valid := TRUE;
    GVL_RECOVERY_REACTIVATION_CONTROL_FABRIC.Recovery_Reactivation_Control_Granted := TRUE;
    GVL_RECOVERY_REACTIVATION_CONTROL_FABRIC.Recovery_Reactivation_Boundary_Stable := TRUE;
    GVL_RECOVERY_REACTIVATION_CONTROL_FABRIC.CrossSubsystem_Reactivation_Consistent := TRUE;
    GVL_RECOVERY_REACTIVATION_CONTROL_FABRIC.Reactivation_Energy_Boundary_Safe := TRUE;
END_IF;
END_PROGRAM

(* ---- PRG_Runtime_Barrier.st ---- *)
PROGRAM PRG_Runtime_Barrier
VAR
    L_Now_MS : UDINT;
    L_Runtime_OK : BOOL := TRUE;
    L_Error_Code : UDINT := 0;
    L_Error_Text : STRING(160) := '';

    L_Finalized_Continuity_Healthy : BOOL;
END_VAR

L_Now_MS := GVL_STATUS.G_System_Time_MS;
L_Runtime_OK := TRUE;
L_Error_Code := 0;
L_Error_Text := '';

// ======================================================
// AUTHORITATIVE RUNTIME BARRIER
// ======================================================
// Creates authoritative runtime publication semantics.
// Rejects impossible runtime states before physical publication.
//
// Runtime authority remains:
// - monotonic-time authoritative;
// - PLC fencing authoritative;
// - transport freshness authoritative.
//
// Distributed finalized continuity now additionally
// participates in primordial runtime authority.
// ======================================================

GVL_RUNTIME_EPOCH.Runtime_Cycle_Start_MS := L_Now_MS;
GVL_RUNTIME_EPOCH.Runtime_Snapshot_Published := FALSE;
GVL_RUNTIME_EPOCH.Runtime_Impossible_State_Detected := FALSE;
GVL_RUNTIME_EPOCH.Runtime_IO_Publication_Allowed := FALSE;

// ------------------------------------------------------
// Monotonic time authority validation.
// ------------------------------------------------------

IF NOT GVL_TIME_MONOTONIC.Monotonic_Time_Initialized THEN
    L_Runtime_OK := FALSE;
    L_Error_Code := 4900;
    L_Error_Text := 'Monotonic time not initialized';
END_IF;

IF L_Runtime_OK AND (NOT GVL_TIME_MONOTONIC.Monotonic_Time_Valid) THEN
    L_Runtime_OK := FALSE;
    L_Error_Code := 4901;
    L_Error_Text := 'Monotonic time invalid';
END_IF;

IF L_Runtime_OK AND GVL_TIME_MONOTONIC.Startup_Quarantine_Active THEN
    L_Runtime_OK := FALSE;
    L_Error_Code := 4902;
    L_Error_Text := 'Startup quarantine active';
END_IF;

IF L_Runtime_OK AND GVL_TIME_MONOTONIC.Time_Rollback_Detected THEN
    L_Runtime_OK := FALSE;
    L_Error_Code := 4903;
    L_Error_Text := 'Monotonic rollback detected';
END_IF;

IF L_Runtime_OK AND GVL_TIME_MONOTONIC.Retained_Time_Invalid THEN
    L_Runtime_OK := FALSE;
    L_Error_Code := 4904;
    L_Error_Text := 'Retained monotonic time invalid';
END_IF;

IF L_Runtime_OK AND (GVL_TIME_MONOTONIC.Boot_Generation_ID = 0) THEN
    L_Runtime_OK := FALSE;
    L_Error_Code := 4905;
    L_Error_Text := 'Boot generation missing';
END_IF;

// ------------------------------------------------------
// Base PLC/runtime authority validation.
// ------------------------------------------------------

IF L_Runtime_OK AND (NOT GVL_STATUS.G_Is_Active_PLC) THEN
    L_Runtime_OK := FALSE;
    L_Error_Code := 5000;
    L_Error_Text := 'Runtime barrier inactive PLC';
END_IF;

// ------------------------------------------------------
// PLC fencing authority validation.
// ------------------------------------------------------

IF L_Runtime_OK AND (NOT GVL_PLC_FENCING.PLC_Ownership_Valid) THEN
    L_Runtime_OK := FALSE;
    L_Error_Code := 5010;
    L_Error_Text := 'PLC ownership invalid';
END_IF;

IF L_Runtime_OK AND (NOT GVL_PLC_FENCING.PLC_Semantic_Authority_Valid) THEN
    L_Runtime_OK := FALSE;
    L_Error_Code := 5011;
    L_Error_Text := 'PLC semantic authority invalid';
END_IF;

IF L_Runtime_OK AND GVL_PLC_FENCING.PLC_Forced_Safe_Quarantine THEN
    L_Runtime_OK := FALSE;
    L_Error_Code := 5012;
    L_Error_Text := 'PLC fencing quarantine active';
END_IF;

IF L_Runtime_OK AND GVL_PLC_FENCING.PLC_Lease_Expired THEN
    L_Runtime_OK := FALSE;
    L_Error_Code := 5013;
    L_Error_Text := 'PLC authority lease expired';
END_IF;

IF L_Runtime_OK AND (GVL_PLC_FENCING.PLC_Fencing_Token = 0) THEN
    L_Runtime_OK := FALSE;
    L_Error_Code := 5014;
    L_Error_Text := 'PLC fencing token missing';
END_IF;

// ------------------------------------------------------
// Transport freshness validation.
// ------------------------------------------------------

IF L_Runtime_OK AND (NOT GVL_TRANSPORT_FRESHNESS.Transport_Freshness_Valid) THEN
    L_Runtime_OK := FALSE;
    L_Error_Code := 5200;
    L_Error_Text := 'Transport freshness invalid';
END_IF;

IF L_Runtime_OK AND (NOT GVL_TRANSPORT_FRESHNESS.Transport_Publication_Allowed) THEN
    L_Runtime_OK := FALSE;
    L_Error_Code := 5201;
    L_Error_Text := 'Transport publication blocked';
END_IF;

IF L_Runtime_OK AND GVL_TRANSPORT_FRESHNESS.Transport_Quarantine_Active THEN
    L_Runtime_OK := FALSE;
    L_Error_Code := 5202;
    L_Error_Text := 'Transport quarantine active';
END_IF;

IF L_Runtime_OK AND GVL_TRANSPORT_FRESHNESS.Transport_Lease_Expired THEN
    L_Runtime_OK := FALSE;
    L_Error_Code := 5203;
    L_Error_Text := 'Transport lease expired';
END_IF;

IF L_Runtime_OK AND GVL_TRANSPORT_FRESHNESS.Transport_Snapshot_Invalid THEN
    L_Runtime_OK := FALSE;
    L_Error_Code := 5204;
    L_Error_Text := 'Transport snapshot invalid';
END_IF;

// ------------------------------------------------------
// Finalized continuity linkage.
// ------------------------------------------------------

L_Finalized_Continuity_Healthy :=
    GVL_SEMANTIC_PROGRESS.Semantic_Forward_Progress_Valid
    AND GVL_SEMANTIC_PROGRESS.Semantic_Execution_Continuity_OK
    AND NOT GVL_SEMANTIC_PROGRESS.Semantic_Progress_Lease_Expired
    AND NOT GVL_SEMANTIC_PROGRESS.Semantic_Progress_Quarantine_Active
    AND GVL_DISTRIBUTED_SNAPSHOT.Distributed_Publication_Reconciled
    AND GVL_DISTRIBUTED_SNAPSHOT.Distributed_Publication_Freeze_Valid
    AND GVL_DISTRIBUTED_SNAPSHOT.Distributed_Snapshot_Consistent
    AND GVL_DISTRIBUTED_COMMIT.Distributed_Commit_Valid
    AND GVL_DISTRIBUTED_COMMIT.Publication_Prepare_Valid
    AND GVL_DISTRIBUTED_COMMIT.Publication_Commit_Confirmed
    AND NOT GVL_DISTRIBUTED_COMMIT.Peer_Commit_Mismatch
    AND NOT GVL_DISTRIBUTED_COMMIT.Commit_Lease_Expired;

IF L_Runtime_OK
AND NOT L_Finalized_Continuity_Healthy THEN
    L_Runtime_OK := FALSE;
    L_Error_Code := 5300;
    L_Error_Text := 'Finalized continuity invalid';
END_IF;

// ------------------------------------------------------
// Impossible-state rejection.
// ------------------------------------------------------

IF L_Runtime_OK THEN
    IF (GVL_SAFETY_SHUTDOWN.G_Safety_Mode = FIRE)
    AND (GVL_COMMAND_SHADOW.G_Vent_Stop)
    THEN
        L_Runtime_OK := FALSE;
        L_Error_Code := 5003;
        L_Error_Text := 'Impossible fire ventilation state';
    END_IF;
END_IF;

IF L_Runtime_OK THEN
    IF (GVL_SAFETY_SHUTDOWN.G_Safety_Mode = GAS)
    AND (NOT GVL_COMMAND_SHADOW.G_Gas_Valve_Close)
    THEN
        L_Runtime_OK := FALSE;
        L_Error_Code := 5004;
        L_Error_Text := 'Impossible gas valve state';
    END_IF;
END_IF;

// ------------------------------------------------------
// Authoritative runtime publication.
// ------------------------------------------------------

GVL_RUNTIME_EPOCH.Runtime_Runtime_Barrier_OK := L_Runtime_OK;
GVL_RUNTIME_EPOCH.Runtime_Snapshot_Valid := L_Runtime_OK;
GVL_RUNTIME_EPOCH.Runtime_PLC_Authority_Valid :=
    GVL_STATUS.G_Is_Active_PLC
    AND GVL_PLC_FENCING.PLC_Semantic_Authority_Valid
    AND GVL_PLC_FENCING.PLC_Ownership_Valid
    AND GVL_TIME_MONOTONIC.Monotonic_Time_Valid
    AND GVL_TRANSPORT_FRESHNESS.Transport_Freshness_Valid
    AND L_Finalized_Continuity_Healthy;

GVL_RUNTIME_EPOCH.Runtime_Last_Validation_Time_MS := L_Now_MS;

IF L_Runtime_OK THEN
    GVL_RUNTIME_EPOCH.Runtime_Epoch := GVL_RUNTIME_EPOCH.Runtime_Epoch + 1;
    GVL_RUNTIME_EPOCH.Runtime_IO_Publication_Allowed := TRUE;
    GVL_RUNTIME_EPOCH.Runtime_Snapshot_Published := TRUE;
    GVL_RUNTIME_EPOCH.Runtime_Last_Error_Code := 0;
    GVL_RUNTIME_EPOCH.Runtime_Last_Error_Text := '';
ELSE
    GVL_RUNTIME_EPOCH.Runtime_Impossible_State_Detected := TRUE;
    GVL_RUNTIME_EPOCH.Runtime_Last_Error_Code := L_Error_Code;
    GVL_RUNTIME_EPOCH.Runtime_Last_Error_Text := L_Error_Text;
    GVL_RUNTIME_EPOCH.Runtime_Barrier_Block_Count := GVL_RUNTIME_EPOCH.Runtime_Barrier_Block_Count + 1;
END_IF;

GVL_RUNTIME_EPOCH.Runtime_Cycle_End_MS := L_Now_MS;
END_PROGRAM

(* ---- PRG_Runtime_Core_Domain.st ---- *)
PROGRAM PRG_Runtime_Core_Domain
// CANONICAL EXECUTION DOMAIN
// PRESERVES EXECUTION ORDER

PRG_Time_Service();
PRG_System_Init();
PRG_Runtime_Barrier();
PRG_Runtime_Snapshot_Governor();
PRG_Runtime_Assumption_Integrity_Governor();

END_PROGRAM

(* ---- PRG_Runtime_IO_Validation.st ---- *)
PROGRAM PRG_Runtime_IO_Validation
VAR
    L_i : INT;
    L_Any_Exhaust_On : BOOL;
    L_Any_Supply_On : BOOL;
    L_Any_Heating_Output_On : BOOL;
    L_Any_Water_Zone_On : BOOL;
    L_Any_Access_Output_On : BOOL;
    L_Any_Lighting_Output_On : BOOL;
    L_Any_Socket_On : BOOL;
    L_Any_Freeze_Circulation_On : BOOL;
    L_Fire_Access_Valid : BOOL;
    L_Water_Leak_Close_Valid : BOOL;
END_VAR

GVL_RUNTIME_IO_VALIDATION.G_Last_Update_MS := GVL_TIME_SERVICE.G_Now_MS;
GVL_RUNTIME_IO_VALIDATION.G_Validation_Executed := TRUE;
GVL_RUNTIME_IO_VALIDATION.G_Validation_Valid := TRUE;

L_Any_Exhaust_On := FALSE;
L_Any_Supply_On := FALSE;
L_Any_Heating_Output_On := FALSE;
L_Any_Water_Zone_On := FALSE;
L_Any_Access_Output_On := FALSE;
L_Any_Lighting_Output_On := FALSE;
L_Any_Socket_On := FALSE;
L_Any_Freeze_Circulation_On := FALSE;
L_Fire_Access_Valid := TRUE;
L_Water_Leak_Close_Valid := TRUE;

FOR L_i := 1 TO GVL_CONSTANTS.C_MAX_EXHAUST_FANS DO
    IF GVL_IO.AO_Exhaust_Fans[L_i] > 0 THEN
        L_Any_Exhaust_On := TRUE;
    END_IF;
END_FOR;

FOR L_i := 1 TO GVL_CONSTANTS.C_MAX_SUPPLY_FANS DO
    IF GVL_IO.AO_Supply_Fans[L_i] > 0 THEN
        L_Any_Supply_On := TRUE;
    END_IF;
END_FOR;

FOR L_i := 1 TO GVL_CONSTANTS.C_MAX_HEATING_CIRCUITS DO
    IF GVL_IO.DO_Zone_Valves[L_i] THEN
        L_Any_Heating_Output_On := TRUE;
    END_IF;
END_FOR;

FOR L_i := 1 TO GVL_CONSTANTS.C_MAX_MANIFOLDS DO
    IF GVL_IO.DO_Manifold_Pumps[L_i] OR (GVL_IO.AO_Manifold_Valves[L_i] > 0) THEN
        L_Any_Heating_Output_On := TRUE;
        L_Any_Freeze_Circulation_On := TRUE;
    END_IF;
END_FOR;

IF GVL_IO.DO_DHW_Heating_Pump
   OR GVL_IO.DO_DHW_Circ_Pump
   OR GVL_IO.DO_Backup_Circulation_Pump
   OR GVL_IO.DO_Electric_Heater_Enable THEN
    L_Any_Heating_Output_On := TRUE;
END_IF;

IF GVL_IO.DO_Backup_Circulation_Pump THEN
    L_Any_Freeze_Circulation_On := TRUE;
END_IF;

FOR L_i := 1 TO GVL_CONSTANTS.C_MAX_WATER_ZONES DO
    IF GVL_IO.DO_Water_Zone_Enable[L_i] THEN
        L_Any_Water_Zone_On := TRUE;
    END_IF;
END_FOR;

L_Any_Access_Output_On :=
    GVL_IO.DO_Gate_Open
    OR GVL_IO.DO_Wicket_Open
    OR GVL_IO.DO_Lock_1_Open
    OR GVL_IO.DO_Lock_1_Close
    OR GVL_IO.DO_Lock_2_Open
    OR GVL_IO.DO_Lock_2_Close;

IF GVL_COMMAND_SHADOW.G_Lock_1_Open AND NOT GVL_IO.DO_Lock_1_Open THEN
    L_Fire_Access_Valid := FALSE;
END_IF;
IF GVL_COMMAND_SHADOW.G_Lock_2_Open AND NOT GVL_IO.DO_Lock_2_Open THEN
    L_Fire_Access_Valid := FALSE;
END_IF;
IF GVL_COMMAND_SHADOW.G_Gate_Open AND NOT GVL_IO.DO_Gate_Open THEN
    L_Fire_Access_Valid := FALSE;
END_IF;
IF GVL_COMMAND_SHADOW.G_Wicket_Open AND NOT GVL_IO.DO_Wicket_Open THEN
    L_Fire_Access_Valid := FALSE;
END_IF;

FOR L_i := 1 TO GVL_CONSTANTS.C_MAX_LIGHT_ZONES DO
    IF GVL_IO.AO_Lighting_Levels[L_i] > 0 THEN
        L_Any_Lighting_Output_On := TRUE;
    END_IF;
END_FOR;

FOR L_i := 1 TO GVL_CONSTANTS.C_MAX_SOCKETS DO
    IF GVL_IO.DO_Sockets[L_i] THEN
        L_Any_Socket_On := TRUE;
    END_IF;
END_FOR;

IF GVL_SAFETY_SHUTDOWN.G_Safety_Mode = WATER_LEAK THEN
    // Four leak zones: 1..3 local pairs, 4 common inlet 35/36.
    IF GVL_INTENT_SAFETY.I_Water_Zone_Close_Required[1] THEN
        L_Water_Leak_Close_Valid :=
            L_Water_Leak_Close_Valid
            AND GVL_IO.DO_Water_Local_Valve_Close[1]
            AND GVL_IO.DO_Water_Local_Valve_Close[2];
    END_IF;

    IF GVL_INTENT_SAFETY.I_Water_Zone_Close_Required[2] THEN
        L_Water_Leak_Close_Valid :=
            L_Water_Leak_Close_Valid
            AND GVL_IO.DO_Water_Local_Valve_Close[3]
            AND GVL_IO.DO_Water_Local_Valve_Close[4];
    END_IF;

    IF GVL_INTENT_SAFETY.I_Water_Zone_Close_Required[3] THEN
        L_Water_Leak_Close_Valid :=
            L_Water_Leak_Close_Valid
            AND GVL_IO.DO_Water_Local_Valve_Close[5]
            AND GVL_IO.DO_Water_Local_Valve_Close[6];
    END_IF;

    IF GVL_INTENT_SAFETY.I_Water_Zone_Close_Required[4]
       OR GVL_INTENT_SAFETY.I_Water_Main_Close_Required
       OR GVL_COMMAND_SHADOW.G_Close_Valve_35
       OR GVL_COMMAND_SHADOW.G_Close_Valve_36 THEN
        L_Water_Leak_Close_Valid :=
            L_Water_Leak_Close_Valid
            AND GVL_IO.DO_Water_Valve_35_Close
            AND GVL_IO.DO_Water_Valve_36_Close;
    END_IF;
END_IF;

GVL_RUNTIME_IO_VALIDATION.Fire_IO_Valid :=
    (NOT GVL_STATUS.G_Is_Active_PLC)
    OR (GVL_SAFETY_SHUTDOWN.G_Safety_Mode <> FIRE)
    OR (
        L_Any_Exhaust_On
        AND NOT L_Any_Supply_On
        AND L_Fire_Access_Valid
    );

GVL_RUNTIME_IO_VALIDATION.Gas_IO_Valid :=
    (NOT GVL_STATUS.G_Is_Active_PLC)
    OR (GVL_SAFETY_SHUTDOWN.G_Safety_Mode <> GAS)
    OR (
        GVL_IO.DO_Gas_Valve_Close
        AND (L_Any_Exhaust_On OR L_Any_Supply_On)
        AND NOT GVL_IO.DO_DHW_Heating_Pump
    );

GVL_RUNTIME_IO_VALIDATION.Leak_IO_Valid :=
    (NOT GVL_STATUS.G_Is_Active_PLC)
    OR (GVL_SAFETY_SHUTDOWN.G_Safety_Mode <> WATER_LEAK)
    OR L_Water_Leak_Close_Valid;

GVL_RUNTIME_IO_VALIDATION.Global_Stop_IO_Valid :=
    (GVL_SAFETY_SHUTDOWN.G_Safety_Mode <> GLOBAL_STOP)
    OR (
        NOT L_Any_Heating_Output_On
        AND NOT L_Any_Exhaust_On
        AND NOT L_Any_Supply_On
        AND NOT L_Any_Water_Zone_On
        AND NOT L_Any_Access_Output_On
        AND NOT L_Any_Lighting_Output_On
        AND NOT L_Any_Socket_On
        AND GVL_IO.DO_Water_Valve_35_Close
        AND GVL_IO.DO_Water_Valve_36_Close
        AND GVL_IO.DO_Gas_Valve_Close
    );

GVL_RUNTIME_IO_VALIDATION.Inactive_PLC_IO_Valid :=
    GVL_STATUS.G_Is_Active_PLC
    OR (
        NOT L_Any_Heating_Output_On
        AND NOT L_Any_Exhaust_On
        AND NOT L_Any_Supply_On
        AND NOT L_Any_Water_Zone_On
        AND NOT L_Any_Access_Output_On
        AND NOT L_Any_Lighting_Output_On
        AND NOT L_Any_Socket_On
        AND GVL_IO.DO_Water_Valve_35_Close
        AND GVL_IO.DO_Water_Valve_36_Close
        AND GVL_IO.DO_Gas_Valve_Close
    );

GVL_RUNTIME_IO_VALIDATION.Freeze_IO_Valid :=
    (NOT GVL_STATUS.G_Is_Active_PLC)
    OR (NOT GVL_STATE.G_Safety_Freeze_Risk)
    OR L_Any_Freeze_Circulation_On;

GVL_RUNTIME_IO_VALIDATION.Any_IO_Invalid :=
    NOT GVL_RUNTIME_IO_VALIDATION.Fire_IO_Valid
    OR NOT GVL_RUNTIME_IO_VALIDATION.Gas_IO_Valid
    OR NOT GVL_RUNTIME_IO_VALIDATION.Leak_IO_Valid
    OR NOT GVL_RUNTIME_IO_VALIDATION.Global_Stop_IO_Valid
    OR NOT GVL_RUNTIME_IO_VALIDATION.Inactive_PLC_IO_Valid
    OR NOT GVL_RUNTIME_IO_VALIDATION.Freeze_IO_Valid;

IF GVL_RUNTIME_IO_VALIDATION.Any_IO_Invalid THEN
    GVL_RUNTIME_IO_VALIDATION.G_Validation_Valid := FALSE;
    GVL_RUNTIME_IO_VALIDATION.Status_Code := 1;
    GVL_RUNTIME_IO_VALIDATION.Status_Text := 'Runtime physical IO validation mismatch';
ELSE
    GVL_RUNTIME_IO_VALIDATION.Status_Code := 0;
    GVL_RUNTIME_IO_VALIDATION.Status_Text := 'Runtime physical IO validation nominal';
END_IF;

// >>> BULK_SYNC_ANCHOR: PRG_Runtime_IO_Validation <<<
END_PROGRAM

(* ---- PRG_Runtime_Scenario_Validation.st ---- *)
PROGRAM PRG_Runtime_Scenario_Validation
// Observational runtime scenario validator.
// Checks that domain execution policy matches current scenario/safety context.
// Does not gate execution and does not write physical outputs.

GVL_RUNTIME_SCENARIO_VALIDATION.G_Last_Update_MS := GVL_TIME_SERVICE.G_Now_MS;
GVL_RUNTIME_SCENARIO_VALIDATION.G_Validation_Executed := TRUE;
GVL_RUNTIME_SCENARIO_VALIDATION.G_Validation_Valid := TRUE;

GVL_RUNTIME_SCENARIO_VALIDATION.Security_Context_Active :=
    GVL_ALARM.G_Security_Armed
    OR GVL_ALARM.G_Security_Alarm;

GVL_RUNTIME_SCENARIO_VALIDATION.Away_Context_Active :=
    GVL_STATUS.G_Current_Scenario = SCENARIO_AWAY;

GVL_RUNTIME_SCENARIO_VALIDATION.Presence_Context_Active :=
    GVL_STATUS.G_Current_Scenario = SCENARIO_PRESENCE;

GVL_RUNTIME_SCENARIO_VALIDATION.Fire_Context_Active :=
    GVL_SAFETY_SHUTDOWN.G_Safety_Mode = FIRE;

GVL_RUNTIME_SCENARIO_VALIDATION.Gas_Context_Active :=
    GVL_SAFETY_SHUTDOWN.G_Safety_Mode = GAS;

GVL_RUNTIME_SCENARIO_VALIDATION.Leak_Context_Active :=
    GVL_SAFETY_SHUTDOWN.G_Safety_Mode = WATER_LEAK;

GVL_RUNTIME_SCENARIO_VALIDATION.Freeze_Context_Active :=
    GVL_STATE.G_Safety_Freeze_Risk
    OR GVL_INPUT.IN_Freeze_Request;

GVL_RUNTIME_SCENARIO_VALIDATION.Heating_Demand_Context_Active :=
    GVL_INPUT.IN_Preheat_Request
    OR GVL_INPUT.IN_Freeze_Request
    OR GVL_HEATING_OUTPUT.DO_DHW_Heating_Pump
    OR GVL_HEATING_OUTPUT.DO_DHW_Circ_Pump
    OR GVL_HEATING_OUTPUT.DO_Backup_Circulation_Pump
    OR GVL_HEATING_OUTPUT.DO_Electric_Heater_Enable;

GVL_RUNTIME_SCENARIO_VALIDATION.Vent_Boost_Context_Active :=
    GVL_INTENT_BEHAVIOR.I_Request_Ventilation_Boost
    OR GVL_COMMAND_SHADOW.G_Vent_PV3_Boost
    OR GVL_COMMAND_SHADOW.G_Exhaust_100_Req
    OR GVL_COMMAND_SHADOW.G_Vent_Smoke_Exhaust;

GVL_RUNTIME_SCENARIO_VALIDATION.Access_Command_Context_Active :=
    GVL_COMMAND_SHADOW.G_Lock_1_Open
    OR GVL_COMMAND_SHADOW.G_Lock_1_Close
    OR GVL_COMMAND_SHADOW.G_Lock_2_Open
    OR GVL_COMMAND_SHADOW.G_Lock_2_Close
    OR GVL_COMMAND_SHADOW.G_Gate_Open
    OR GVL_COMMAND_SHADOW.G_Wicket_Open
    OR GVL_ACCESS_RUNTIME.G_Any_Pulse_Active;

GVL_RUNTIME_SCENARIO_VALIDATION.Idle_Context_Active :=
    NOT GVL_RUNTIME_SCENARIO_VALIDATION.Security_Context_Active
    AND NOT GVL_RUNTIME_SCENARIO_VALIDATION.Away_Context_Active
    AND NOT GVL_RUNTIME_SCENARIO_VALIDATION.Presence_Context_Active
    AND NOT GVL_RUNTIME_SCENARIO_VALIDATION.Fire_Context_Active
    AND NOT GVL_RUNTIME_SCENARIO_VALIDATION.Gas_Context_Active
    AND NOT GVL_RUNTIME_SCENARIO_VALIDATION.Leak_Context_Active
    AND NOT GVL_RUNTIME_SCENARIO_VALIDATION.Freeze_Context_Active
    AND NOT GVL_RUNTIME_SCENARIO_VALIDATION.Heating_Demand_Context_Active
    AND NOT GVL_RUNTIME_SCENARIO_VALIDATION.Vent_Boost_Context_Active
    AND NOT GVL_RUNTIME_SCENARIO_VALIDATION.Access_Command_Context_Active;

GVL_RUNTIME_SCENARIO_VALIDATION.Idle_Context_Valid :=
    (NOT GVL_RUNTIME_SCENARIO_VALIDATION.Idle_Context_Active)
    OR (
        GVL_DOMAIN_EXECUTION_POLICY.Access_Mode = 0
        AND GVL_DOMAIN_EXECUTION_POLICY.Lighting_Mode = 0
        AND GVL_DOMAIN_EXECUTION_POLICY.Water_Mode = 0
        AND GVL_DOMAIN_EXECUTION_POLICY.Heating_Mode = 0
        AND GVL_DOMAIN_EXECUTION_POLICY.Vent_Mode = 0
    );

GVL_RUNTIME_SCENARIO_VALIDATION.Security_Context_Valid :=
    (NOT GVL_RUNTIME_SCENARIO_VALIDATION.Security_Context_Active)
    OR (
        GVL_DOMAIN_EXECUTION_POLICY.Access_Mode >= 1
        AND GVL_DOMAIN_EXECUTION_POLICY.Lighting_Mode >= 1
        AND GVL_DOMAIN_EXECUTION_POLICY.Water_Mode >= 1
    );

GVL_RUNTIME_SCENARIO_VALIDATION.Fire_Context_Valid :=
    (NOT GVL_RUNTIME_SCENARIO_VALIDATION.Fire_Context_Active)
    OR (
        GVL_DOMAIN_EXECUTION_POLICY.Access_Mode = 2
        AND GVL_DOMAIN_EXECUTION_POLICY.Lighting_Mode = 2
        AND GVL_DOMAIN_EXECUTION_POLICY.Vent_Mode = 2
    );

GVL_RUNTIME_SCENARIO_VALIDATION.Gas_Context_Valid :=
    (NOT GVL_RUNTIME_SCENARIO_VALIDATION.Gas_Context_Active)
    OR (
        GVL_DOMAIN_EXECUTION_POLICY.Access_Mode = 2
        AND GVL_DOMAIN_EXECUTION_POLICY.Vent_Mode = 2
        AND GVL_DOMAIN_EXECUTION_POLICY.Heating_Mode = 2
    );

GVL_RUNTIME_SCENARIO_VALIDATION.Leak_Context_Valid :=
    (NOT GVL_RUNTIME_SCENARIO_VALIDATION.Leak_Context_Active)
    OR (GVL_DOMAIN_EXECUTION_POLICY.Water_Mode = 2);

GVL_RUNTIME_SCENARIO_VALIDATION.Freeze_Context_Valid :=
    (NOT GVL_RUNTIME_SCENARIO_VALIDATION.Freeze_Context_Active)
    OR (GVL_DOMAIN_EXECUTION_POLICY.Heating_Mode >= 1);

GVL_RUNTIME_SCENARIO_VALIDATION.Heating_Context_Valid :=
    (NOT GVL_RUNTIME_SCENARIO_VALIDATION.Heating_Demand_Context_Active)
    OR (GVL_DOMAIN_EXECUTION_POLICY.Heating_Mode >= 1);

GVL_RUNTIME_SCENARIO_VALIDATION.Vent_Context_Valid :=
    (NOT GVL_RUNTIME_SCENARIO_VALIDATION.Vent_Boost_Context_Active)
    OR (GVL_DOMAIN_EXECUTION_POLICY.Vent_Mode >= 1);

GVL_RUNTIME_SCENARIO_VALIDATION.Access_Context_Valid :=
    (NOT GVL_RUNTIME_SCENARIO_VALIDATION.Access_Command_Context_Active)
    OR (GVL_DOMAIN_EXECUTION_POLICY.Access_Mode = 2);

GVL_RUNTIME_SCENARIO_VALIDATION.Any_Context_Invalid :=
    NOT GVL_RUNTIME_SCENARIO_VALIDATION.Idle_Context_Valid
    OR NOT GVL_RUNTIME_SCENARIO_VALIDATION.Security_Context_Valid
    OR NOT GVL_RUNTIME_SCENARIO_VALIDATION.Fire_Context_Valid
    OR NOT GVL_RUNTIME_SCENARIO_VALIDATION.Gas_Context_Valid
    OR NOT GVL_RUNTIME_SCENARIO_VALIDATION.Leak_Context_Valid
    OR NOT GVL_RUNTIME_SCENARIO_VALIDATION.Freeze_Context_Valid
    OR NOT GVL_RUNTIME_SCENARIO_VALIDATION.Heating_Context_Valid
    OR NOT GVL_RUNTIME_SCENARIO_VALIDATION.Vent_Context_Valid
    OR NOT GVL_RUNTIME_SCENARIO_VALIDATION.Access_Context_Valid;

IF GVL_RUNTIME_SCENARIO_VALIDATION.Any_Context_Invalid THEN
    GVL_RUNTIME_SCENARIO_VALIDATION.G_Validation_Valid := FALSE;
    GVL_RUNTIME_SCENARIO_VALIDATION.Status_Code := 1;
    GVL_RUNTIME_SCENARIO_VALIDATION.Status_Text := 'Runtime scenario validation mismatch';
ELSE
    GVL_RUNTIME_SCENARIO_VALIDATION.Status_Code := 0;
    GVL_RUNTIME_SCENARIO_VALIDATION.Status_Text := 'Runtime scenario validation nominal';
END_IF;

// >>> BULK_SYNC_ANCHOR: PRG_Runtime_Scenario_Validation <<<
END_PROGRAM

(* ---- PRG_Runtime_Snapshot_Governor.st ---- *)
PROGRAM PRG_Runtime_Snapshot_Governor
VAR
    L_Now_MS : UDINT;
    L_Snapshot_Valid : BOOL := TRUE;
    L_Error_Code : UDINT := 0;
    L_Error_Text : STRING(160) := '';
END_VAR

L_Now_MS := GVL_STATUS.G_System_Time_MS;
L_Snapshot_Valid := TRUE;
L_Error_Code := 0;
L_Error_Text := '';

// ======================================================
// IMMUTABLE RUNTIME SNAPSHOT GOVERNOR
// ======================================================
// Governs immutable publication snapshot semantics.
// Prevents mutable runtime publication leakage.
// ======================================================

GVL_RUNTIME_SNAPSHOT.Snapshot_Mutation_Detected := FALSE;
GVL_RUNTIME_SNAPSHOT.Snapshot_Publication_Allowed := FALSE;
GVL_RUNTIME_SNAPSHOT.Snapshot_Frozen := FALSE;

// Runtime authority linkage.
IF NOT GVL_RUNTIME_EPOCH.Runtime_Runtime_Barrier_OK THEN
    L_Snapshot_Valid := FALSE;
    L_Error_Code := 12000;
    L_Error_Text := 'Runtime authority invalid';
END_IF;

// Observability synchronization linkage.
IF L_Snapshot_Valid
AND (NOT GVL_OBSERVABILITY_AUTHORITY.Authority_Snapshot_Valid)
THEN
    L_Snapshot_Valid := FALSE;
    L_Error_Code := 12001;
    L_Error_Text := 'Observability snapshot invalid';
END_IF;

// Output freshness linkage.
IF L_Snapshot_Valid
AND GVL_OUTPUT_EPOCH.Output_Forced_Safe_Decay
THEN
    L_Snapshot_Valid := FALSE;
    L_Error_Code := 12002;
    L_Error_Text := 'Output decay active';
END_IF;

// Mutation detection foundation.
IF L_Snapshot_Valid
AND GVL_RUNTIME_EPOCH.Runtime_Impossible_State_Detected
THEN
    L_Snapshot_Valid := FALSE;
    L_Error_Code := 12003;
    L_Error_Text := 'Runtime mutation anomaly detected';

    GVL_RUNTIME_SNAPSHOT.Snapshot_Mutation_Detected := TRUE;
END_IF;

// Immutable snapshot freeze semantics.
IF L_Snapshot_Valid THEN
    GVL_RUNTIME_SNAPSHOT.Snapshot_Frozen := TRUE;
    GVL_RUNTIME_SNAPSHOT.Snapshot_Publication_Allowed := TRUE;

    GVL_RUNTIME_SNAPSHOT.Snapshot_Copy_Valid := TRUE;
    GVL_RUNTIME_SNAPSHOT.Snapshot_Isolation_Valid := TRUE;

    GVL_RUNTIME_SNAPSHOT.Snapshot_Runtime_Authority_Valid := TRUE;
    GVL_RUNTIME_SNAPSHOT.Snapshot_Observability_Synchronized := TRUE;

    GVL_RUNTIME_SNAPSHOT.Snapshot_Freeze_Start_MS := L_Now_MS;
    GVL_RUNTIME_SNAPSHOT.Snapshot_Last_Publication_MS := L_Now_MS;

    GVL_RUNTIME_SNAPSHOT.Snapshot_Epoch := GVL_RUNTIME_SNAPSHOT.Snapshot_Epoch + 1;
    GVL_RUNTIME_SNAPSHOT.Snapshot_Publication_Epoch := GVL_RUNTIME_SNAPSHOT.Snapshot_Publication_Epoch + 1;

    GVL_RUNTIME_SNAPSHOT.Snapshot_Last_Error_Code := 0;
    GVL_RUNTIME_SNAPSHOT.Snapshot_Last_Error_Text := '';
ELSE
    GVL_RUNTIME_SNAPSHOT.Snapshot_Frozen := FALSE;
    GVL_RUNTIME_SNAPSHOT.Snapshot_Publication_Allowed := FALSE;

    GVL_RUNTIME_SNAPSHOT.Snapshot_Copy_Valid := FALSE;
    GVL_RUNTIME_SNAPSHOT.Snapshot_Isolation_Valid := FALSE;

    GVL_RUNTIME_SNAPSHOT.Snapshot_Runtime_Authority_Valid := FALSE;
    GVL_RUNTIME_SNAPSHOT.Snapshot_Observability_Synchronized := FALSE;

    GVL_RUNTIME_SNAPSHOT.Snapshot_Last_Error_Code := L_Error_Code;
    GVL_RUNTIME_SNAPSHOT.Snapshot_Last_Error_Text := L_Error_Text;

    GVL_RUNTIME_SNAPSHOT.Snapshot_Invalidation_Count := GVL_RUNTIME_SNAPSHOT.Snapshot_Invalidation_Count + 1;
END_IF;
END_PROGRAM

(* ---- PRG_Runtime_Sustainability_Governor.st ---- *)
PROGRAM PRG_Runtime_Sustainability_Governor
VAR
    L_Now_MS : UDINT;
    L_Runtime_Valid : BOOL := TRUE;
    L_Error_Code : UDINT := 0;
    L_Error_Text : STRING(160) := '';
END_VAR

L_Now_MS := GVL_STATUS.G_System_Time_MS;
L_Runtime_Valid := TRUE;
L_Error_Code := 0;
L_Error_Text := '';

// Fail-safe defaults.
GVL_RUNTIME_SUSTAINABILITY_FABRIC.Runtime_Sustainability_Valid := FALSE;
GVL_RUNTIME_SUSTAINABILITY_FABRIC.Runtime_Sustainability_Granted := FALSE;
GVL_RUNTIME_SUSTAINABILITY_FABRIC.Runtime_Sustainability_Quarantine_Active := TRUE;

GVL_RUNTIME_SUSTAINABILITY_FABRIC.Deterministic_Cycle_Budget_Stable := FALSE;
GVL_RUNTIME_SUSTAINABILITY_FABRIC.Runtime_Queue_Load_Stable := FALSE;
GVL_RUNTIME_SUSTAINABILITY_FABRIC.Memory_Fragmentation_Stable := FALSE;
GVL_RUNTIME_SUSTAINABILITY_FABRIC.Watchdog_Jitter_Stable := FALSE;
GVL_RUNTIME_SUSTAINABILITY_FABRIC.HA_Synchronization_Load_Stable := FALSE;

// Energy causality authority required.
IF NOT GVL_ENERGY_CAUSALITY_FABRIC.Energy_Causality_Granted THEN
    L_Runtime_Valid := FALSE;
    L_Error_Code := 38000;
    L_Error_Text := 'Energy causality authority not granted';
END_IF;

// Resource-collapse detectors.
IF GVL_RUNTIME_SUSTAINABILITY_FABRIC.Memory_Fragmentation_Drift_Detected THEN
    L_Runtime_Valid := FALSE;
    L_Error_Code := 38001;
    L_Error_Text := 'Memory fragmentation drift detected';
END_IF;

IF GVL_RUNTIME_SUSTAINABILITY_FABRIC.Queue_Saturation_Detected THEN
    L_Runtime_Valid := FALSE;
    L_Error_Code := 38002;
    L_Error_Text := 'Runtime queue saturation detected';
END_IF;

IF GVL_RUNTIME_SUSTAINABILITY_FABRIC.Historical_Persistence_Amplification_Detected THEN
    L_Runtime_Valid := FALSE;
    L_Error_Code := 38003;
    L_Error_Text := 'Historical persistence amplification detected';
END_IF;

IF GVL_RUNTIME_SUSTAINABILITY_FABRIC.Watchdog_Jitter_Escalation_Detected THEN
    L_Runtime_Valid := FALSE;
    L_Error_Code := 38004;
    L_Error_Text := 'Watchdog jitter escalation detected';
END_IF;

IF GVL_RUNTIME_SUSTAINABILITY_FABRIC.HASynchronization_Overload_Detected THEN
    L_Runtime_Valid := FALSE;
    L_Error_Code := 38005;
    L_Error_Text := 'HA synchronization overload detected';
END_IF;

IF GVL_RUNTIME_SUSTAINABILITY_FABRIC.Deterministic_Cycle_Erosion_Detected THEN
    L_Runtime_Valid := FALSE;
    L_Error_Code := 38006;
    L_Error_Text := 'Deterministic cycle erosion detected';
END_IF;

// Long-term runtime sustainability validation.
IF L_Runtime_Valid
AND NOT GVL_RUNTIME_SUSTAINABILITY_FABRIC.Historical_Persistence_Load_Stable THEN
    L_Runtime_Valid := FALSE;
    L_Error_Code := 38010;
    L_Error_Text := 'Historical persistence load unstable';
END_IF;

IF L_Runtime_Valid
AND NOT GVL_RUNTIME_SUSTAINABILITY_FABRIC.Snapshot_Publication_Stable THEN
    L_Runtime_Valid := FALSE;
    L_Error_Code := 38011;
    L_Error_Text := 'Snapshot publication unstable';
END_IF;

IF L_Runtime_Valid
AND NOT GVL_RUNTIME_SUSTAINABILITY_FABRIC.Distributed_Runtime_Load_Coherent THEN
    L_Runtime_Valid := FALSE;
    L_Error_Code := 38012;
    L_Error_Text := 'Distributed runtime load coherence invalid';
END_IF;

IF L_Runtime_Valid
AND NOT GVL_RUNTIME_SUSTAINABILITY_FABRIC.Runtime_Evolution_Sustainable THEN
    L_Runtime_Valid := FALSE;
    L_Error_Code := 38013;
    L_Error_Text := 'Runtime evolution sustainability invalid';
END_IF;

IF L_Runtime_Valid THEN
    GVL_RUNTIME_SUSTAINABILITY_FABRIC.Runtime_Sustainability_Valid := TRUE;
    GVL_RUNTIME_SUSTAINABILITY_FABRIC.Runtime_Sustainability_Granted := TRUE;
    GVL_RUNTIME_SUSTAINABILITY_FABRIC.Runtime_Sustainability_Quarantine_Active := FALSE;

    GVL_RUNTIME_SUSTAINABILITY_FABRIC.Deterministic_Cycle_Budget_Stable := TRUE;
    GVL_RUNTIME_SUSTAINABILITY_FABRIC.Runtime_Queue_Load_Stable := TRUE;
    GVL_RUNTIME_SUSTAINABILITY_FABRIC.Memory_Fragmentation_Stable := TRUE;
    GVL_RUNTIME_SUSTAINABILITY_FABRIC.Watchdog_Jitter_Stable := TRUE;
    GVL_RUNTIME_SUSTAINABILITY_FABRIC.HA_Synchronization_Load_Stable := TRUE;

    GVL_RUNTIME_SUSTAINABILITY_FABRIC.Runtime_Sustainability_Epoch :=
        GVL_ENERGY_CAUSALITY_FABRIC.Energy_Causality_Epoch;

    GVL_RUNTIME_SUSTAINABILITY_FABRIC.Runtime_Sustainability_Epoch_Coherent := TRUE;

    GVL_RUNTIME_SUSTAINABILITY_FABRIC.Runtime_Sustainability_Last_Update_MS :=
        L_Now_MS;

    GVL_RUNTIME_SUSTAINABILITY_FABRIC.Runtime_Sustainability_Lease_Expired := FALSE;

    GVL_RUNTIME_SUSTAINABILITY_FABRIC.Runtime_Sustainability_Last_Error_Code := 0;
    GVL_RUNTIME_SUSTAINABILITY_FABRIC.Runtime_Sustainability_Last_Error_Text := '';
ELSE
    GVL_RUNTIME_SUSTAINABILITY_FABRIC.Runtime_Sustainability_Valid := FALSE;
    GVL_RUNTIME_SUSTAINABILITY_FABRIC.Runtime_Sustainability_Granted := FALSE;
    GVL_RUNTIME_SUSTAINABILITY_FABRIC.Runtime_Sustainability_Quarantine_Active := TRUE;

    GVL_RUNTIME_SUSTAINABILITY_FABRIC.Runtime_Sustainability_Lease_Expired := TRUE;

    GVL_RUNTIME_SUSTAINABILITY_FABRIC.Runtime_Sustainability_Last_Error_Code :=
        L_Error_Code;

    GVL_RUNTIME_SUSTAINABILITY_FABRIC.Runtime_Sustainability_Last_Error_Text :=
        L_Error_Text;

    GVL_RUNTIME_SUSTAINABILITY_FABRIC.Runtime_Sustainability_Invalidation_Count :=
        GVL_RUNTIME_SUSTAINABILITY_FABRIC.Runtime_Sustainability_Invalidation_Count + 1;
END_IF;

END_PROGRAM

(* ---- PRG_Runtime_Transition_Validator.st ---- *)
PROGRAM PRG_Runtime_Transition_Validator
// PASSIVE FORMAL TRANSITION VALIDATOR
// NO EXECUTION MUTATION
// NO AUTHORITY MUTATION
// OBSERVABILITY ONLY

GVL_RUNTIME_TRANSITION_SYSTEM.Runtime_Transition_Legal := FALSE;
GVL_RUNTIME_TRANSITION_SYSTEM.Runtime_Transition_Proofs_Valid := FALSE;
GVL_RUNTIME_TRANSITION_SYSTEM.Runtime_Transition_Lineage_Valid := FALSE;
GVL_RUNTIME_TRANSITION_SYSTEM.Runtime_Transition_Temporal_Valid := FALSE;

CASE GVL_RUNTIME_STATE_ALGEBRA.Current_Runtime_State OF

    SYS_SAFE:
        GVL_RUNTIME_TRANSITION_SYSTEM.Runtime_Transition_Legal := TRUE;
        GVL_RUNTIME_TRANSITION_SYSTEM.Runtime_Transition_Proofs_Valid := TRUE;

    SYS_RECOVERING:
        GVL_RUNTIME_TRANSITION_SYSTEM.Runtime_Transition_Legal :=
            GVL_TEMPORAL_CAUSALITY_CLOSURE_FABRIC.Temporal_Causality_Coherent;

        GVL_RUNTIME_TRANSITION_SYSTEM.Runtime_Transition_Proofs_Valid :=
            GVL_SAFETY_OBSERVABILITY_TRUTH_FABRIC.Observability_Reality_Equivalence_Granted;

        GVL_RUNTIME_TRANSITION_SYSTEM.Runtime_Transition_Lineage_Valid :=
            GVL_AUTHORITY_LINEAGE_FABRIC.Authority_Lineage_Valid;

        GVL_RUNTIME_TRANSITION_SYSTEM.Runtime_Transition_Temporal_Valid :=
            GVL_DISTRIBUTED_EPOCH_LINEARITY_FABRIC.Epoch_Timeline_Monotonic;

    SYS_QUARANTINED:
        GVL_RUNTIME_TRANSITION_SYSTEM.Runtime_Transition_Legal := TRUE;

    SYS_TRUSTLESS:
        GVL_RUNTIME_TRANSITION_SYSTEM.Runtime_Transition_Legal := FALSE;
        GVL_RUNTIME_TRANSITION_SYSTEM.Unsafe_Trust_Escalation_Observed := TRUE;

ELSE
    GVL_RUNTIME_TRANSITION_SYSTEM.Illegal_Runtime_Transition_Observed := TRUE;

END_CASE;

END_PROGRAM

(* ---- PRG_Safety.st ---- *)
PROGRAM PRG_Safety
VAR
    fbWaterLeakageManager : FB_Water_Leakage_Manager;
    fbGasSmokeManager : FB_Gas_Smoke_Manager;
    fbOwnership : FB_Ownership_Watchdog;
    L_i : INT;
END_VAR

GVL_INTENT_SAFETY.I_Source_Valid := TRUE;
GVL_INTENT_SAFETY.I_Last_Update_MS := GVL_TIME_SERVICE.G_Now_MS;
GVL_INTENT_SAFETY.I_Fire_Alarm_Active := FALSE;
GVL_INTENT_SAFETY.I_Gas_Alarm_Active := FALSE;
GVL_INTENT_SAFETY.I_Leak_Alarm_Active := FALSE;
GVL_INTENT_SAFETY.I_CO_Warning_Active := FALSE;
GVL_INTENT_SAFETY.I_System_Safe_Stop_Required := FALSE;
GVL_INTENT_SAFETY.I_Freeze_Protection_Required := FALSE;
GVL_INTENT_SAFETY.I_Evacuation_Mode_Active := FALSE;
GVL_INTENT_SAFETY.I_Gas_Close_Required := FALSE;
GVL_INTENT_SAFETY.I_Boiler_Stop_Required := FALSE;
GVL_INTENT_SAFETY.I_Vent_Stop_Required := FALSE;
GVL_INTENT_SAFETY.I_Vent_Force_PV3_Boost := FALSE;
GVL_INTENT_SAFETY.I_Vent_Force_Supply_100 := FALSE;
GVL_INTENT_SAFETY.I_Vent_Force_Supply_80 := FALSE;
GVL_INTENT_SAFETY.I_Vent_Force_Exhaust_100 := FALSE;
GVL_INTENT_SAFETY.I_Water_Main_Close_Required := FALSE;
GVL_INTENT_SAFETY.I_Water_Selective_Recovery_Allowed := FALSE;
GVL_INTENT_SAFETY.I_Water_Recovery_Target_Zone := 0;
FOR L_i := 1 TO 32 DO
    GVL_INTENT_SAFETY.I_Water_Zone_Close_Required[L_i] := FALSE;
END_FOR;
GVL_INTENT_SAFETY.I_Lock_1_Force_Open := FALSE;
GVL_INTENT_SAFETY.I_Lock_1_Force_Close_Block := FALSE;
GVL_INTENT_SAFETY.I_Lock_2_Force_Open := FALSE;
GVL_INTENT_SAFETY.I_Lock_2_Force_Close_Block := FALSE;
GVL_INTENT_SAFETY.I_Test_Timeout_Gas_Close := FALSE;
GVL_INTENT_SAFETY.I_Test_Timeout_Water_Close := FALSE;

fbWaterLeakageManager(
    VI_System_Time_MS := GVL_TIME_SERVICE.G_Now_MS,
    VI_IsActivePLC := GVL_STATUS.G_Is_Active_PLC,
    VI_Sensors := GVL_STATE.G_Water_Sensors,
    VI_Config := GVL_CONFIG.G_HMI_Flood_Config,
    VO_Status_Msg => GVL_STATUS.G_Flood_Status_Msg,
    VO_Leak_Detected => GVL_HEALTH_BRIDGE.G_Leak_Detected,
    VO_Leak_Warning_Level => GVL_HEALTH_BRIDGE.G_Leak_Warning_Level
);
GVL_INTENT_SAFETY.I_Leak_Alarm_Active := GVL_HEALTH_BRIDGE.G_Leak_Detected;
GVL_INTENT_SAFETY.I_Water_Main_Close_Required := GVL_HEALTH_BRIDGE.G_Leak_Detected;

fbGasSmokeManager(
    VI_System_Time_MS := GVL_TIME_SERVICE.G_Now_MS,
    VI_IsActivePLC := GVL_STATUS.G_Is_Active_PLC,
    VI_Methane_LEL := GVL_Safety_Selector.G_Methane_Effective_Array,
    VI_CO_PPM := GVL_Safety_Selector.G_CO_Effective_Array,
    VI_Smoke_Sensors := GVL_Safety_Selector.G_Smoke_Effective_Array,
    VI_Mute_Request := GVL_CONFIG.G_HMI_Mute_Alarm,
    VO_Smoke_Detected => GVL_HEALTH_BRIDGE.G_Smoke_Detected,
    VO_Gas_Detected => GVL_HEALTH_BRIDGE.G_Gas_Detected,
    VO_Methane_Warning_Level => GVL_HEALTH_BRIDGE.G_Methane_Warning_Level,
    VO_Methane_Alarm_Level => GVL_HEALTH_BRIDGE.G_Methane_Alarm_Level,
    VO_Methane_Critical_Level => GVL_HEALTH_BRIDGE.G_Methane_Critical_Level,
    VO_CO_Warning_Level => GVL_HEALTH_BRIDGE.G_CO_Warning_Level,
    VO_CO_Alarm_Level => GVL_HEALTH_BRIDGE.G_CO_Alarm_Level,
    VO_Status_Msg => GVL_STATUS.G_Gas_Status_Msg
);

GVL_INTENT_SAFETY.I_Fire_Alarm_Active := GVL_HEALTH_BRIDGE.G_Smoke_Detected;
GVL_INTENT_SAFETY.I_Gas_Alarm_Active :=
    GVL_HEALTH_BRIDGE.G_Methane_Alarm_Level
    OR GVL_HEALTH_BRIDGE.G_Methane_Critical_Level
    OR GVL_HEALTH_BRIDGE.G_CO_Alarm_Level;
GVL_INTENT_SAFETY.I_CO_Warning_Active := GVL_HEALTH_BRIDGE.G_CO_Warning_Level;

// Methane 10% LEL warning: ventilation boost only.
IF GVL_HEALTH_BRIDGE.G_Methane_Warning_Level THEN
    GVL_INTENT_SAFETY.I_Vent_Force_PV3_Boost := TRUE;
END_IF;

// Methane 20% LEL alarm or CO alarm: close gas and stop boilers.
IF GVL_HEALTH_BRIDGE.G_Methane_Alarm_Level OR
   GVL_HEALTH_BRIDGE.G_Methane_Critical_Level OR
   GVL_HEALTH_BRIDGE.G_CO_Alarm_Level THEN
    GVL_INTENT_SAFETY.I_Gas_Close_Required := TRUE;
    GVL_INTENT_SAFETY.I_Boiler_Stop_Required := TRUE;
END_IF;

// Methane 40% LEL critical: full escalation.
IF GVL_HEALTH_BRIDGE.G_Methane_Critical_Level THEN
    GVL_INTENT_SAFETY.I_System_Safe_Stop_Required := TRUE;
    GVL_INTENT_SAFETY.I_Evacuation_Mode_Active := TRUE;
    GVL_INTENT_SAFETY.I_Vent_Force_Supply_100 := TRUE;
END_IF;

// Ownership watchdog must observe authoritative safety truth, not stale
// projected GVL_STATE.G_Safety_*_Alarm compatibility fields.
fbOwnership(
    VI_Gas_Level := GVL_Safety_Selector.G_Methane_Effective_Array[GVL_CONSTANTS.C_PRIMARY_EFFECTIVE_GAS_INDEX],
    VI_Gas_Alarm := GVL_INTENT_SAFETY.I_Gas_Alarm_Active,
    VI_Leak_Alarm := GVL_HEALTH_BRIDGE.G_Leak_Detected,
    VI_Smoke_Alarm := GVL_HEALTH_BRIDGE.G_Smoke_Detected
);

IF fbOwnership.VO_Ownership_Violation THEN
    GVL_DEBUG_VIEW.D_Ownership_Violation := TRUE;
END_IF;

IF GVL_STATE.G_Safety_Smoke_Latched THEN
    GVL_INTENT_SAFETY.I_System_Safe_Stop_Required := TRUE;
    GVL_INTENT_SAFETY.I_Evacuation_Mode_Active := TRUE;
    GVL_INTENT_SAFETY.I_Boiler_Stop_Required := TRUE;
    GVL_INTENT_SAFETY.I_Vent_Stop_Required := TRUE;
    GVL_INTENT_SAFETY.I_Lock_1_Force_Open := TRUE;
    GVL_INTENT_SAFETY.I_Lock_1_Force_Close_Block := TRUE;
    GVL_INTENT_SAFETY.I_Lock_2_Force_Open := TRUE;
    GVL_INTENT_SAFETY.I_Lock_2_Force_Close_Block := TRUE;
END_IF;

IF GVL_STATE.G_Safety_Gas_Latched THEN
    GVL_INTENT_SAFETY.I_System_Safe_Stop_Required := TRUE;
    GVL_INTENT_SAFETY.I_Gas_Close_Required := TRUE;
    GVL_INTENT_SAFETY.I_Boiler_Stop_Required := TRUE;
    GVL_INTENT_SAFETY.I_Vent_Force_PV3_Boost := TRUE;
    GVL_INTENT_SAFETY.I_Vent_Force_Supply_100 := TRUE;
END_IF;

IF GVL_HEALTH_BRIDGE.G_CO_Warning_Level OR GVL_HEALTH_BRIDGE.G_CO_Alarm_Level THEN
    GVL_INTENT_SAFETY.I_Vent_Force_Supply_80 := TRUE;
END_IF;

IF GVL_STATE.G_Safety_Leak_Latched THEN
    GVL_INTENT_SAFETY.I_Water_Main_Close_Required := TRUE;
END_IF;

IF GVL_STATUS.G_Diagnostics.Water_Main_Shutdown_Recommended OR
   GVL_STATUS.G_Diagnostics.Water_Close_Fault_Active THEN
    GVL_INTENT_SAFETY.I_Water_Main_Close_Required := TRUE;
    GVL_INTENT_SAFETY.I_Leak_Alarm_Active := TRUE;
END_IF;

IF GVL_STATE.G_Freeze_Hardware_Degraded THEN
    GVL_INTENT_SAFETY.I_Freeze_Protection_Required := TRUE;
END_IF;

// >>> BULK_SYNC_ANCHOR: PRG_Safety <<<
END_PROGRAM

(* ---- PRG_Safety_Observability_Truth_Governor.st ---- *)
PROGRAM PRG_Safety_Observability_Truth_Governor
IF GVL_DISTRIBUTED_FORWARD_PROGRESS_FABRIC.Distributed_Forward_Progress_Granted
AND NOT GVL_SAFETY_OBSERVABILITY_TRUTH_FABRIC.FakeSafe_Projection_Detected
AND NOT GVL_SAFETY_OBSERVABILITY_TRUTH_FABRIC.Telemetry_Reality_Divergence_Detected
AND NOT GVL_SAFETY_OBSERVABILITY_TRUTH_FABRIC.Stale_Safety_Projection_Detected
AND NOT GVL_SAFETY_OBSERVABILITY_TRUTH_FABRIC.Safety_Observability_Fork_Detected THEN

    GVL_SAFETY_OBSERVABILITY_TRUTH_FABRIC.Safety_Observability_Truth_Valid := TRUE;
    GVL_SAFETY_OBSERVABILITY_TRUTH_FABRIC.Safety_Observability_Truth_Granted := TRUE;
    GVL_SAFETY_OBSERVABILITY_TRUTH_FABRIC.Safety_Reality_Projection_Valid := TRUE;
    GVL_SAFETY_OBSERVABILITY_TRUTH_FABRIC.Observability_Reality_Equivalence_Granted := TRUE;
    GVL_SAFETY_OBSERVABILITY_TRUTH_FABRIC.Physical_Safety_Projection_Canonical := TRUE;
END_IF;
END_PROGRAM

(* ---- PRG_Safety_Operator.st ---- *)
PROGRAM PRG_Safety_Operator
VAR
    fbSafetyWorkflow : FB_Safety_Workflow_Manager;
END_VAR

// Operator / test / recover workflow ownership.

fbSafetyWorkflow(
    VI_System_Time_MS := GVL_TIME_SERVICE.G_Now_MS,
    VI_Water_Selective_Recover := GVL_INTENT_USER.I_Water_Selective_Recover,
    VI_Gas_Selective_Recover := GVL_INTENT_USER.I_Gas_Selective_Recover,
    VI_Water_Valve_Test_Open := GVL_INTENT_USER.I_Water_Valve_Test_Open,
    VI_Water_Valve_Test_Close := GVL_INTENT_USER.I_Water_Valve_Test_Close,
    VI_Water_Valve_Test_Confirm := GVL_INTENT_USER.I_Water_Valve_Test_Confirm,
    VI_Gas_Valve_Test_Open := GVL_INTENT_USER.I_Gas_Valve_Test_Open,
    VI_Gas_Valve_Test_Close := GVL_INTENT_USER.I_Gas_Valve_Test_Close,
    VI_Gas_Valve_Test_Confirm := GVL_INTENT_USER.I_Gas_Valve_Test_Confirm
);

// selective recover requests enter the deterministic recovery state machine
IF fbSafetyWorkflow.VO_Water_Selective_Recover_Edge OR
   fbSafetyWorkflow.VO_Gas_Selective_Recover_Edge THEN
    GVL_SAFETY_RECOVERY.G_Recovery_Requested := TRUE;
END_IF;

// propagate test timeout safety actions
IF fbSafetyWorkflow.VO_Water_Test_Timeout_Close_Required THEN
    GVL_INTENT_SAFETY.I_Test_Timeout_Water_Close := TRUE;
END_IF;

IF fbSafetyWorkflow.VO_Gas_Test_Timeout_Close_Required THEN
    GVL_INTENT_SAFETY.I_Test_Timeout_Gas_Close := TRUE;
END_IF;

// move recovery manual confirm here
IF GVL_INTENT_USER.I_Reset_Errors THEN
    GVL_SAFETY_RECOVERY.G_Recovery_Manual_Confirm := TRUE;
END_IF;

// >>> BULK_SYNC_ANCHOR: PRG_Safety_Operator <<<
END_PROGRAM

(* ---- PRG_Safety_Recovery.st ---- *)
PROGRAM PRG_Safety_Recovery
VAR
    L_Phase : E_Recovery_Phase;
    L_Mode_Active : BOOL;
    L_Time_OK : BOOL;
END_VAR

L_Mode_Active := GVL_SAFETY_SHUTDOWN.G_Safety_Active;
L_Phase := GVL_SAFETY_RECOVERY.G_Recovery_Phase;

CASE L_Phase OF

    IDLE:
        IF NOT L_Mode_Active AND GVL_SAFETY_RECOVERY.G_Recovery_Requested THEN
            GVL_SAFETY_RECOVERY.G_Recovery_Phase := STABILIZING;
            GVL_SAFETY_RECOVERY.G_Recovery_Active := TRUE;
            GVL_SAFETY_RECOVERY.G_Recovery_Start_MS := GVL_TIME_SERVICE.G_Now_MS;
            GVL_SAFETY_RECOVERY.G_Recovery_Abort_Reason := 0;
        END_IF;

    STABILIZING:
        IF L_Mode_Active THEN
            GVL_SAFETY_RECOVERY.G_Recovery_Phase := ABORTED;
            GVL_SAFETY_RECOVERY.G_Recovery_Abort_Reason := 1;
        ELSIF (GVL_TIME_SERVICE.G_Now_MS - GVL_SAFETY_RECOVERY.G_Recovery_Start_MS) > GVL_SAFETY_RECOVERY_CONFIG.G_Stabilization_Delay_MS THEN
            GVL_SAFETY_RECOVERY.G_Recovery_Phase := WAIT_MANUAL_CONFIRM;
            GVL_SAFETY_RECOVERY.G_Recovery_Stable_Since_MS := GVL_TIME_SERVICE.G_Now_MS;
        END_IF;

    WAIT_MANUAL_CONFIRM:
        IF L_Mode_Active THEN
            GVL_SAFETY_RECOVERY.G_Recovery_Phase := ABORTED;
            GVL_SAFETY_RECOVERY.G_Recovery_Abort_Reason := 1;
        ELSIF GVL_SAFETY_RECOVERY.G_Recovery_Manual_Confirm THEN
            GVL_SAFETY_RECOVERY.G_Recovery_Phase := RECOVERING;
        END_IF;

    RECOVERING:
        IF L_Mode_Active THEN
            GVL_SAFETY_RECOVERY.G_Recovery_Phase := ABORTED;
            GVL_SAFETY_RECOVERY.G_Recovery_Abort_Reason := 1;
        ELSE
            GVL_SAFETY_RECOVERY.G_Recovery_Phase := COOLDOWN;
            GVL_SAFETY_RECOVERY.G_Recovery_Cooldown_Start_MS := GVL_TIME_SERVICE.G_Now_MS;
        END_IF;

    COOLDOWN:
        IF L_Mode_Active THEN
            GVL_SAFETY_RECOVERY.G_Recovery_Phase := ABORTED;
            GVL_SAFETY_RECOVERY.G_Recovery_Abort_Reason := 1;
        ELSE
            L_Time_OK := (GVL_TIME_SERVICE.G_Now_MS - GVL_SAFETY_RECOVERY.G_Recovery_Cooldown_Start_MS) > GVL_SAFETY_RECOVERY_CONFIG.G_Cooldown_Time_MS;

            IF L_Time_OK THEN
                GVL_SAFETY_RECOVERY.G_Recovery_Phase := IDLE;
                GVL_SAFETY_RECOVERY.G_Recovery_Active := FALSE;
                GVL_SAFETY_RECOVERY.G_Recovery_Requested := FALSE;
                GVL_SAFETY_RECOVERY.G_Recovery_Manual_Confirm := FALSE;
            END_IF;
        END_IF;

    ABORTED:
        GVL_SAFETY_RECOVERY.G_Recovery_Active := FALSE;
        GVL_SAFETY_RECOVERY.G_Recovery_Requested := FALSE;
        GVL_SAFETY_RECOVERY.G_Recovery_Manual_Confirm := FALSE;
        IF NOT L_Mode_Active THEN
            GVL_SAFETY_RECOVERY.G_Recovery_Phase := IDLE;
        END_IF;

END_CASE;

END_PROGRAM
// >>> BULK_SYNC_ANCHOR: PRG_Safety_Recovery <<<

(* ---- PRG_Safety_Shutdown.st ---- *)
PROGRAM PRG_Safety_Shutdown
VAR
    L_Mode : E_Safety_Mode := NORMAL;
END_VAR

// Input degraded forces safe stop first
IF GVL_INPUT.IN_Input_Degraded THEN
    L_Mode := GLOBAL_STOP;
ELSE

    // Priority: FIRE > GAS > WATER > GLOBAL_STOP > NORMAL

    IF GVL_INTENT_SAFETY.I_Fire_Alarm_Active THEN
        L_Mode := FIRE;
    ELSIF GVL_INTENT_SAFETY.I_Gas_Close_Required OR GVL_INTENT_SAFETY.I_Test_Timeout_Gas_Close THEN
        L_Mode := GAS;
    ELSIF GVL_INTENT_SAFETY.I_Leak_Alarm_Active OR
          GVL_INTENT_SAFETY.I_Water_Main_Close_Required OR
          GVL_INTENT_SAFETY.I_Test_Timeout_Water_Close THEN
        L_Mode := WATER_LEAK;
    ELSIF GVL_INTENT_SAFETY.I_System_Safe_Stop_Required THEN
        L_Mode := GLOBAL_STOP;
    ELSE
        L_Mode := NORMAL;
    END_IF;

END_IF;

GVL_SAFETY_SHUTDOWN.G_Safety_Mode := L_Mode;
GVL_SAFETY_SHUTDOWN.G_Safety_Active := (L_Mode <> NORMAL);

// >>> BULK_SYNC_ANCHOR: PRG_Safety_Shutdown <<<
END_PROGRAM
